Universal Robots URScript: 127765-201_OpticalBench_V1.script

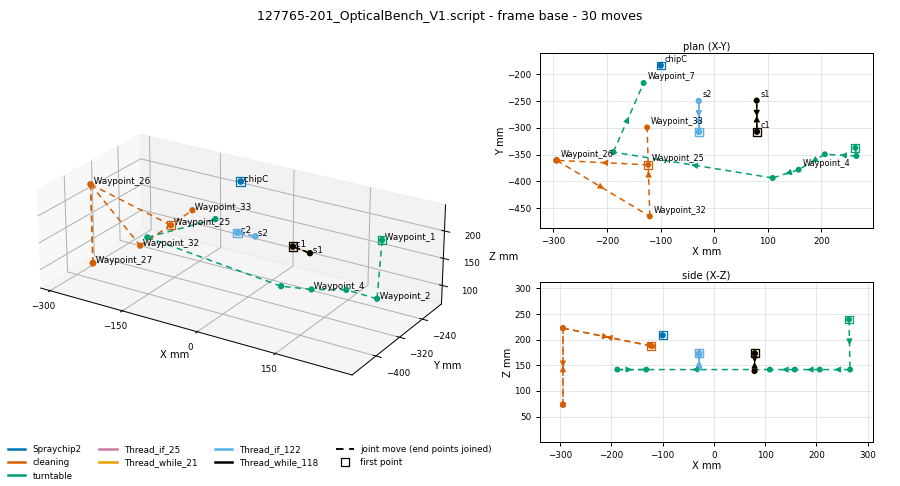
[picture p0: tool path of 127765-201_OpticalBench_V1.script in frame base, 30 of 121 moves have a stored position in this frame; points joined in program order, loops and branches not executed]
def P127765201_OpticalBench_V1():
  global _hidden_verificationVariable=0
  step_count_28707e12_0c2a_4f39_b822_8a6eb026eba7 = 0.0
  thread Step_Counter_Thread_bc455d1c_3720_4032_8e16_f4a00f067eee():
    while (True):
      step_count_28707e12_0c2a_4f39_b822_8a6eb026eba7 = step_count_28707e12_0c2a_4f39_b822_8a6eb026eba7 + 1.0
      sync()
    end
  end
  run Step_Counter_Thread_bc455d1c_3720_4032_8e16_f4a00f067eee()
  set_target_payload(0.530000, [0.009000, -0.039000, 0.092000], [0.000534, 0.000534, 0.000534, 0.000000, 0.000000, 0.000000])
  set_safety_mode_transition_hardness(1)
  set_tcp(p[0.0,0.0,0.11,0.0,0.0,0.0])
  set_tool_communication(False, 115200, 0, 1, 1.5, 3.5)
  set_tool_output_mode(0)
  set_tool_digital_output_mode(0, 1)
  set_tool_digital_output_mode(1, 1)
  set_tool_voltage(0)
  set_gravity([0.0, 0.0, 9.82])
  set_standard_analog_input_domain(0, 1)
  set_standard_analog_input_domain(1, 1)
  set_tool_analog_input_domain(0, 1)
  set_tool_analog_input_domain(1, 1)
  set_analog_outputdomain(0, 0)
  set_analog_outputdomain(1, 0)
  set_input_actions_to_default()
  global Al_plate=p[0.12405209206180495,-0.2666666051843552,0.020008101224669964,-9.276623980477388E-5,1.8107917580596192E-5,3.1233857134705927]
  global Frame2x2=p[0.18266245434305164,-0.34273121659514855,0.026002571110600767,-2.225423529876215E-4,3.0110667546023537E-4,3.1233976058306383]
  global Plane_1=p[0.0,0.0,0.0,0.0,0.0,0.0]
  global URlogoTutorial=p[-0.08178353973148575,-0.3363174165299142,0.04788621506469384,-3.9746155723688456E-5,-3.4682148779121894E-5,-1.5668291789091222]
  global carousel=p[0.13865255139760183,-0.25132593351268107,0.051531504137083003,-4.453572132438073E-5,-1.3071222590669835E-4,-3.1349676625391965]
  global carouselrod=p[0.2020731702281844,-0.34951442511341274,0.1947611446273096,3.139766958234101,-0.10689428010274801,-1.1796370330365635E-5]
  global paper=p[-0.09670794781244417,-0.3283412964648025,0.027665994240809913,-3.2057893450593004E-5,2.867088716161181E-5,-1.6085327915291054]
  global rod=p[0.13368013097420872,-0.41123185103490206,0.09926814901395645,2.2214229924093103,-2.2214158162465862,-2.9165882738638143E-5]
  # begin: URCap Installation Node
  #   Source: Remote TCP & Toolpath, 1.3.0.build16, Universal Robots A/S
  #   Type: Remote TCP & Toolpath
  mc_check_divergence = True
  mc_lookahead = 0.03
  mc_gain = 2000
  mc_dt = 0.004

  mc_conv_tol_s = 0.001
  mc_conv_loops = 100

  mc_ee_set_id = 2

  MC_GROUP_STANDBY = 0
  MC_GROUP_STOPPING = 2
  MC_GROUP_ERROR_STOP = 3

  MC_ERROR_PATHDIVERGED = 0
  MC_ERROR_COLLISION = 1
  MC_ERROR_JOINTLIMIT = 2
  MC_ERROR_SINGULARITY = 4
  MC_ERROR_PLANNINGFAILED = 16
  MC_ERROR_DAEMONSTOPPED = 1024
  MC_ERROR_SERVER_BUSY = 1025
  MC_ERROR_NOT_INITIALIZED = 2000

  MC_TOOLPATH_ERROR_NONE = 0
  MC_TOOLPATH_ERROR_FILELOAD = 1
  MC_TOOLPATH_ERROR_PARSE = 2
  MC_TOOLPATH_ERROR_EMPTYTOOLPATH = 3
  MC_TOOLPATH_ERROR_UNSUPPORTEDTYPE = 4

  MC_GROUP_STATUS_INPUT = 24
  MC_CURRENT_MOTION_ID_INPUT = 25
  MC_ERROR_CODE_INPUT = 26
  MC_DIGITAL_OUTPUTS_INPUT = 27
  MC_JOINT_VALUE_INPUT = 24
  MC_WATCHDOG_INPUT = 30
  MC_PATH_SPEED_INPUT = 31
  MC_SPEEDFACTOR_OUTPUT = 24

  mc_last_watchdog = 0
  mc_watchdog_counter = 0
  mc_watchdog_counter_limit = 100

  mc_last_motion_id = -1
  mc_group_status = MC_GROUP_STOPPING
  mc_server_started = False
  mc_rtcp_moving = False
  mc_debug_msg = False
  mc_gmm_initialized = False
  mc_last_digital_outputs = 0

  def mc_initialize(mode, tcp, doc=6):
  	mc_check_busy()

  	if (mode == 0 and doc == 6):
  		mc_ee_set_id = 0
  	end

  	if (mode == 1 and doc == 6):
  		mc_ee_set_id = 2
  	end

  	if (mode == 0 and doc == 5):
  		mc_ee_set_id = 1
  	end

  	if (mode == 1 and doc == 5):
  		mc_ee_set_id = 3
  	end

  	mc_initialize_internal(tcp)
  end

  def mc_initialize_internal(tcp):
  	if (mc_server_started == False):
  		global mc_server = rpc_factory("xmlrpc", "127.0.0.1:7828")
  		mc_server_started = True
  	end

  	mc_server.setDataStoreBoolean("IS_ON", "/robot/check_divergence", mc_check_divergence)
  	mc_server.reset()
  	mc_group_status = MC_GROUP_STANDBY
  	mc_set_speed_factor(1.0)
  	mc_server.setKinTransform(mc_ee_set_id, 0, tcp)
  	mc_gmm_initialized = False
  end

  def mc_check_busy():
  	enter_critical
  	if (mc_rtcp_moving == False):
  		mc_rtcp_moving = True
  	else:
  		mc_error_stop("", "", MC_ERROR_SERVER_BUSY)
  	end
  	exit_critical
  end

  def mc_add_linear(pose, a, v, r):
  	mc_check_ready()
  	ee_id = 0
  	buffer_mode = "BLENDING_NEXT"
  	transition_mode = "CORNER_DISTANCE"
  	id = mc_server.moveLinearAbsolute(pose, mc_ee_set_id, ee_id, v, a, buffer_mode, transition_mode, r)

  	if (id == -1):
  		mc_error_stop("Compute node returned ID ", id)
  	end

  	mc_last_motion_id = id

  	return id
  end

  def mc_add_circular(pose_via, pose_to, a, v, r, mode = 0):
  	mc_check_ready()
  	ee_id = 0
  	buffer_mode = "BLENDING_NEXT"
  	transition_mode = "CORNER_DISTANCE"
  	id = mc_server.moveCircularBorderAbsolute(pose_via, pose_to, mode, mc_ee_set_id, ee_id, v, a, buffer_mode, transition_mode, r)

  	if (id == -1):
  		mc_error_stop("Compute node returned ID ", id)
  	end

  	mc_last_motion_id = id

  	return id
  end

  def mc_add_path(path_id, a, v, r):
  	mc_check_ready()
  	ee_id = 0
  	buffer_mode = "BLENDING_NEXT"
  	transition_mode = "CORNER_DISTANCE"
  	id = mc_server.movePath(path_id, mc_ee_set_id, ee_id, v, a, buffer_mode, transition_mode, r)

  	if (id == -1):
  		result = mc_server.getErrorCode()
  		mc_toolpath_error_stop(result[0], result[1])
  	end

  	mc_last_motion_id = id

  	return id
  end

  def mc_load_path(nc_file, use_feedrate = False):
  	id = mc_server.loadPath(nc_file, use_feedrate)

  	if (id < 0):
  		result = mc_server.getErrorCode()
  		mc_toolpath_error_stop(result[0], result[1])
  	end

  	return id
  end

  def mc_get_target_rtcp_speed():
  	return read_input_float_register(MC_PATH_SPEED_INPUT)
  end

  def mc_check_ready():
  	if mc_group_status != MC_GROUP_STANDBY:
  		mc_error_stop("", "", MC_ERROR_NOT_INITIALIZED)
  	end
  end

  def mc_set_pcs(pcs):
  	ee_id = 0
  	mc_server.setCoordinateTransform(mc_ee_set_id, ee_id, pcs, "ABORTING")
  end

  def mc_set_digital_outputs():
  	current_do = read_input_integer_register(MC_DIGITAL_OUTPUTS_INPUT)
  	current_do_bin = integer_to_binary_list(current_do)
  	last_do_bin = integer_to_binary_list(mc_last_digital_outputs)
  	loopcounter = 0
  	while (loopcounter < 4):
  		value_bit = loopcounter * 6
  		port_bit_0 = value_bit + 1
  		port_bit_1 = value_bit + 2
  		port_bit_2 = value_bit + 3
  		port_bit_3 = value_bit + 4
  		port_bit_4 = value_bit + 5
  		last_port = binary_list_to_integer([last_do_bin[port_bit_0], last_do_bin[port_bit_1], last_do_bin[port_bit_2], last_do_bin[port_bit_3], last_do_bin[port_bit_4]])
  		current_port = binary_list_to_integer([current_do_bin[port_bit_0], current_do_bin[port_bit_1], current_do_bin[port_bit_2], current_do_bin[port_bit_3], current_do_bin[port_bit_4]])
  		if (current_port != 0 and (current_port != last_port or current_do_bin[value_bit] != last_do_bin[value_bit])):
  			if (current_port <= 8):
  				set_standard_digital_out(current_port - 1, current_do_bin[value_bit])
  			elif (current_port <= 16):
  				set_configurable_digital_out(current_port - 9, current_do_bin[value_bit])
  			else:
  				set_tool_digital_out(current_port - 17, current_do_bin[value_bit])
  			end
  		end
  		loopcounter = loopcounter + 1
  	end
  	mc_last_digital_outputs = current_do
  end

  def mc_run_motion(id=-1):
  	if (id == -1):
  		id = mc_last_motion_id
  	end

  	mc_debugMsg("Waiting for ID ", id)

  	if (mc_gmm_initialized == False):
  		mc_initialize_gmm()
  	end

  	mc_current_motion_id = read_input_integer_register(MC_CURRENT_MOTION_ID_INPUT)
  	mc_group_status = read_input_integer_register(MC_GROUP_STATUS_INPUT)
  	joint_targets = get_actual_joint_positions()
  	while (mc_current_motion_id <= id and mc_current_motion_id != -2 and mc_group_status != MC_GROUP_STOPPING and mc_group_status != MC_GROUP_ERROR_STOP):
  		mc_current_motion_id = read_input_integer_register(MC_CURRENT_MOTION_ID_INPUT)
  		mc_group_status = read_input_integer_register(MC_GROUP_STATUS_INPUT)

  		joint_targets = mc_get_joint_targets(joint_targets)
  		servoj(joint_targets, t = mc_dt, lookahead_time = mc_lookahead, gain = mc_gain)

  		mc_set_digital_outputs()

  		mc_check_watchdog()
  	end

  	if (mc_group_status == MC_GROUP_STOPPING or mc_group_status == MC_GROUP_ERROR_STOP):
  		stopj(45)

  		mc_debugMsg("Stopping due to error after ID ", id)

  		mc_server.setDataStoreBoolean("IS_RTCP_RUNNING", "/group_motion_manager", False)

  		error_code = read_input_integer_register(MC_ERROR_CODE_INPUT)
  		mc_error_stop("Compute node returned group status ", mc_group_status, error_code)

  		mc_rtcp_moving = False
  		mc_group_status = MC_GROUP_STOPPING
  	end

  	if (id == mc_last_motion_id):
  		mc_debugMsg("Stopping after ID ", id)
  		mc_check_convergence(joint_targets)

  		mc_server.setDataStoreBoolean("IS_RTCP_RUNNING", "/group_motion_manager", False)

  		mc_rtcp_moving = False
  		mc_group_status = MC_GROUP_STOPPING
  	end

  	mc_debugMsg("Completed ID ", id)
  end

  def mc_set_speed_factor(s):
  	write_output_float_register(MC_SPEEDFACTOR_OUTPUT, s)
  end

  def mc_initialize_gmm():
  	mc_current_motion_id = read_input_integer_register(MC_CURRENT_MOTION_ID_INPUT)
  	while (mc_current_motion_id != -1):
  		mc_current_motion_id = read_input_integer_register(MC_CURRENT_MOTION_ID_INPUT)
  		sleep(mc_dt)
  		mc_check_watchdog()
  	end

  	mc_server.setDataStoreBoolean("IS_RTCP_RUNNING", "/group_motion_manager", True)

  	while (mc_current_motion_id == -1):
  		mc_current_motion_id = read_input_integer_register(MC_CURRENT_MOTION_ID_INPUT)
  		sleep(mc_dt)
  		mc_check_watchdog()
  	end

  	mc_gmm_initialized = True
  end

  def mc_check_convergence(joint_targets):
  	loopcounter = 0
  	converged = False
  	while (converged == False and loopcounter < mc_conv_loops):

  		joint_targets = mc_get_joint_targets(joint_targets)
  		ur_targets = get_target_joint_positions()
  		joint_speeds = get_actual_joint_speeds()

  		position_converged = joint_targets[0] == ur_targets[0] and joint_targets[1] == ur_targets[1] and joint_targets[2] == ur_targets[2] and joint_targets[3] == ur_targets[3] and joint_targets[4] == ur_targets[4] and joint_targets[5] == ur_targets[5]
  		speed_converged = joint_speeds[0] <= mc_conv_tol_s and joint_speeds[1] <= mc_conv_tol_s and joint_speeds[2] <= mc_conv_tol_s and joint_speeds[3] <= mc_conv_tol_s and joint_speeds[4] <= mc_conv_tol_s and joint_speeds[5] <= mc_conv_tol_s
  		converged = position_converged and speed_converged

  		servoj(joint_targets, t = mc_dt, lookahead_time = mc_lookahead, gain = mc_gain)

  		loopcounter = loopcounter + 1
  	end

  	mc_debugMsg("Convergence loop count: ", loopcounter)
  end

  def mc_check_watchdog():
  	current_watchdog = read_input_float_register(MC_WATCHDOG_INPUT)

  	if (current_watchdog > mc_last_watchdog):
  		mc_last_watchdog = current_watchdog
  		mc_watchdog_counter = 0
  	else:
  		mc_watchdog_counter = mc_watchdog_counter + 1
  		if (mc_watchdog_counter > mc_watchdog_counter_limit):
  			mc_error_stop("", "", MC_ERROR_DAEMONSTOPPED)
  		end
  	end
  end

  def mc_get_joint_targets(joint_targets):
  	joint_targets[0] = read_input_float_register(MC_JOINT_VALUE_INPUT)
  	joint_targets[1] = read_input_float_register(MC_JOINT_VALUE_INPUT + 1)
  	joint_targets[2] = read_input_float_register(MC_JOINT_VALUE_INPUT + 2)
  	joint_targets[3] = read_input_float_register(MC_JOINT_VALUE_INPUT + 3)
  	joint_targets[4] = read_input_float_register(MC_JOINT_VALUE_INPUT + 4)
  	joint_targets[5] = read_input_float_register(MC_JOINT_VALUE_INPUT + 5)
  	return joint_targets
  end

  def mc_error_stop(msg, param="", error_code=MC_ERROR_PLANNINGFAILED):
  	if (msg != ""):
  		textmsg(msg, param)
  	end

  	textmsg("Error code: ", error_code)
  	error_msg = mc_getErrorMessage(error_code)
  	textmsg(error_msg)

  	popup(error_msg, title="Remote TCP", error=True, blocking=False)
  	halt
  end

  def mc_toolpath_error_stop(error_code, param):
  	msg = mc_getToolpathMessage(error_code)
  	textmsg(msg + " - Line: ", param)

  	popup(msg, title="Toolpath Validation", error=True, blocking=True)
  	halt
  end

  def mc_debugMsg(msg, param=""):
  	if (mc_debug_msg == True):
  		textmsg(msg, param)
  	end
  end
  def mc_getErrorMessage(error_code):
  	if error_code == MC_ERROR_PATHDIVERGED:
  		return "<html>Robot cannot maintain tool speed. You may avoid this issue by:<ul><li>reducing the tool speed;</li><li>avoiding sharp corners;</li><li>staying away from singularities.</li></ul></html>"
  	elif error_code == MC_ERROR_COLLISION:
  		return "Robot is in collision."
  	elif error_code == MC_ERROR_JOINTLIMIT:
  		return "Robot is at a joint limit."
  	elif error_code == MC_ERROR_SINGULARITY:
  		return "Robot is at a singularity."
  	elif error_code == MC_ERROR_DAEMONSTOPPED:
  		return "The controller stopped."
  	elif error_code == MC_ERROR_SERVER_BUSY:
  		return "Another Remote TCP Move node is running."
  	elif error_code == MC_ERROR_NOT_INITIALIZED:
  		return "Group motion manager is not initialized."
  	else:
  		return "Motion planning failed."
  	end
  end

  def mc_getToolpathMessage(message_code):
  	if message_code == MC_TOOLPATH_ERROR_NONE:
  		return "Toolpath file is valid."
  	elif message_code == MC_TOOLPATH_ERROR_FILELOAD:
  		return "File cannot be loaded."
  	elif message_code == MC_TOOLPATH_ERROR_PARSE:
  		return "Parsing error"
  	elif message_code == MC_TOOLPATH_ERROR_EMPTYTOOLPATH:
  		return "Empty toolpath"
  	elif message_code == MC_TOOLPATH_ERROR_UNSUPPORTEDTYPE:
  		return "Unsupported type"
  	else:
  		return "Unknown toolpath validation error"
  	end
  end
  # end: URCap Installation Node
  # begin: URCap Installation Node
  #   Source: Robotiq_Copilot, 2.7.0.56387, Robotiq Inc.
  #   Type: Machine Tending
  def rq_is_stack_light_machine_state_running():
    return False
  end
  def rq_is_stack_light_machine_state_idle():
    return False
  end
  # end: URCap Installation Node
  # begin: URCap Installation Node
  #   Source: Robotiq_Copilot, 2.7.0.56387, Robotiq Inc.
  #   Type: Copilot
  ###############################################################
  # Script file used to communicate with Robotiq's ft sensor
  # Version: 0.0.1
  ###############################################################

  node_rpc_server = rpc_factory("xmlrpc","http://127.0.0.1:4251/node")
  linalg = rpc_factory("xmlrpc","http://127.0.0.1:4251/linalg")
  storevar = rpc_factory("xmlrpc","http://127.0.0.1:4251/storevariable")
  kinematics_rpc_server = rpc_factory("xmlrpc","http://127.0.0.1:4251/")

  global Fx = 0.0
  global Fy = 0.0
  global Fz = 0.0
  global Mx = 0.0
  global My = 0.0
  global Mz = 0.0
  global T_base_sensor = p[0,0,0,0,0,0]
  global tcp_wrench = [0,0,0,0,0,0]
  global base_wrench = [0,0,0,0,0,0]
  global sensor_wrench = [0,0,0,0,0,0]
  global rq_depal_end_pose_offset = p[0,0,0,0,0,0]
  global rq_ft_sensor_connected = False

  rq_target_joint_positions = get_actual_joint_positions()
  rq_elapsed_time = 0
  rq_force_protect_urcap = 0.0
  rq_torque_protect_urcap = 0.0
  rq_collision_detection_enabled = False
  rq_collision_detection_active_time = 0.0
  rq_halt_on_collision_detection = True
  is_rq_prevent_steady_enabled = True
  rq_active_node = 0
  rq_node_executor_thread_running = False
  rq_lookahead_time = 0.05
  rq_continue_node_execution = True
  rq_controller_time_step = 0.008

  rq_linear_axis_move_abs_target_position = 0.0
  rq_linear_axis_move_abs_target_speed = 0.0 # Documented in monorepo/doc/pal/PalAdvancedProgrammingFunctions.md
  rq_linear_axis_move_abs_target_acc = 0.0 # Documented in monorepo/doc/pal/PalAdvancedProgrammingFunctions.md
  rq_linear_axis_move_abs_target_decel = 0.0 # Documented in monorepo/doc/pal/PalAdvancedProgrammingFunctions.md
  rq_linear_axis_move_absolute_thread = 0
  rq_linear_axis_move_absolute_thread_running = False

  def pose_to_list(p):
    return [p[0], p[1], p[2], p[3], p[4], p[5]]
  end

  def list_to_pose(l):
    return p[l[0], l[1], l[2], l[3], l[4], l[5]]
  end

  def rq_init_path(pathId):
     initPathAnswer = node_rpc_server.initpath(pathId)
     verify_path_answer(initPathAnswer)
     return initPathAnswer[0]
  end

  def concat(str1, str2, str3):
    return str_cat(str1, str_cat(str2, str3))
  end
  def key_val(key, val):
    return concat(concat("`", key, "`"), ":", val)
  end

  thread rq_prevent_steady():
    local q_start = get_target_joint_positions()
    local q = q_start
    local p = 0

    while True:
      p = p + rq_controller_time_step*4*3.14159
      local offset = 0.000001*sin(p)
      q[5] = q_start[5] + offset
      servoj(q)
    end
  end

  def linear_axis_move_abs(target_position,
                           target_speed,
                           target_acceleration,
                           target_deceleration,
                           is_blocking,
                           prevent_steady = True):
    rq_linear_axis_move_abs_target_position = target_position
    rq_linear_axis_move_abs_target_speed = target_speed
    rq_linear_axis_move_abs_target_acc = target_acceleration
    rq_linear_axis_move_abs_target_decel = target_deceleration
    is_rq_prevent_steady_enabled = prevent_steady

    if( rq_linear_axis_move_absolute_thread_running ):
      kill rq_linear_axis_move_absolute_thread
    end
    rq_linear_axis_move_absolute_thread = run linear_axis_move_abs_thread()
    if(is_blocking):
      join rq_linear_axis_move_absolute_thread
    end
  end #linear_axis_move_abs

  thread linear_axis_move_abs_thread():

    if is_rq_prevent_steady_enabled:
      rq_prevent_steady_thread = run rq_prevent_steady()
    end

    rq_linear_axis_move_absolute_thread_running = True
    timeout_in_milliseconds = 500
    target_position_reached = False
    number_of_done_status_received_while_not_at_target = 0

    while( not target_position_reached ):
      move_absolute_response = node_rpc_server.linearaxismove(rq_linear_axis_move_abs_target_position,
                                                              rq_linear_axis_move_abs_target_speed,
                                                              rq_linear_axis_move_abs_target_acc,
                                                              rq_linear_axis_move_abs_target_decel,
                                                              timeout_in_milliseconds)

      if move_absolute_response == 0: # Done
        position_tolerance = 1e-3
        local position = node_rpc_server.linearaxisgetactualposition() # local because it is a variable under 15 chars that a user could have defined
        target_position_reached = ( norm( position - rq_linear_axis_move_abs_target_position ) < position_tolerance )
        if not target_position_reached:
          number_of_done_status_received_while_not_at_target = number_of_done_status_received_while_not_at_target + 1
          if ( number_of_done_status_received_while_not_at_target > 10 ): #When the move starts, it may take some time before the status changes from done to busy so we accept a certain number of done status without being at the target position
            textmsg("error: target position should be reached when move absolute status is Done")
          end
        end
      elif move_absolute_response == 1: # Normal (safeguard stopped, busy moving, or paused)
        # do nothing
      elif move_absolute_response == 2: # Error
        textmsg("Linear axis absolute move error")
        popup("Program paused because axis is not ready or the requested position is outside the allowed range.",
              title="Linear axis move error", warning=False, error=True, blocking=True)
        socket_send_line("pause", "RQDashboardClient") # If the axis is not ready, this allows the user to go fix it and then resume the program.
        sleep(1.0) # The socket_send_line command is non-blocking, so we need to wait for the progam to pause.
                   # Without the sleep, execution will continue and multiple popups and program pauses will be executed.
      end

      sleep(rq_controller_time_step)
    end #while
    rq_linear_axis_move_absolute_thread_running = False

    if is_rq_prevent_steady_enabled:
      kill rq_prevent_steady_thread
    end

  end # linear_axis_move_abs_thread

  def setup_force_node_on_server(generic_rq_insertion_force_node_id = 1,
                                 feature=1,
                                 targetforce = [0,0,0,0,0,0],
                                 force_control_enabled_axes = [False, False, False, False, False, False],
                                 max_negative_deviation_vector = [-0.1, -0.1, -0.1, -0.1, -0.1, -0.1],
                                 max_positive_deviation_vector = [0.1, 0.1, 0.1, 0.1, 0.1, 0.1],
                                 adaptiveStiffness = True):
    node_rpc_server.setforcecontrolfeature(generic_rq_insertion_force_node_id, feature)
    node_rpc_server.setforcecontroltargetforce(generic_rq_insertion_force_node_id, targetforce)
    node_rpc_server.setforcecontrolenabledaxes(generic_rq_insertion_force_node_id, force_control_enabled_axes)
    node_rpc_server.setforcecontrolmaximaldeviation(generic_rq_insertion_force_node_id, max_negative_deviation_vector, max_positive_deviation_vector)
    node_rpc_server.setforcecontroladaptivestiffnessenabledaxes(generic_rq_insertion_force_node_id, True)
  end

  def verify_path_answer(path_answer):
   initPathStatusCode = path_answer[1]
   handle_path_node_error_code(initPathStatusCode)
  end

  def handle_path_node_error_code(initPathStatusCode):
    if initPathStatusCode == -1:
      popup("Could not compute path with the selected options.", "Robotiq's FT Sensor", blocking=True, error=True)
    elif initPathStatusCode == 1:
      popup("Joint solution impossible. Change your starting position.", "Robotiq's FT Sensor", blocking=True, error=True)
    elif initPathStatusCode == 2:
      popup("Discontinuous path detected. Change your starting position.", "Robotiq's FT Sensor", blocking=True, error=True)
    elif initPathStatusCode == 3:
      popup("Path time limit has been reached. Increase the speed of your path or break it down in multiple shorter paths.", "Robotiq's FT Sensor", blocking=True, error=True)
    elif initPathStatusCode == 4:
      popup("Could not compute path with the selected options. Computing path timeout.", "Robotiq's FT Sensor", blocking=True, error=True)
    elif initPathStatusCode == 5:
      popup("Path computation was aborted.", "Robotiq's FT Sensor", blocking=True, error=True)
    elif initPathStatusCode == 6:
      popup("A previous path computation is still in progress. Please try again in a few seconds.", "Robotiq's FT Sensor", blocking=True, error=True)
    elif initPathStatusCode == 7:
      textmsg("Path initialization error: Invalid path id.") # No popup needed in this case.
    elif initPathStatusCode == 8:
      popup("Palletizer error: box number out of range.", blocking=True, error=True)
    elif initPathStatusCode == 9:
      popup("Palletizer error: collision detected.", blocking=True, error=True)
    elif initPathStatusCode == 10:
      popup("Palletizer error: boxes overlap in layer.", blocking=True, error=True)
    elif initPathStatusCode == 11:
      popup("Palletizer error: empty layer.", blocking=True, error=True)
    elif initPathStatusCode == 12:
      popup("Palletizer error: The PLC was not connected during node creation.", blocking=True, error=True)
    elif initPathStatusCode != 0:
      textmsg("Unexpected initPathStatusCode value : ", initPathStatusCode)
    end

    if initPathStatusCode != 0:
      halt
    end
  end

  def rq_wait_ft_sensor_steady(timeout = 2000):

    max_mean_squared_error = [0.1, 0.1, 0.1, 0.0001, 0.0001, 0.0001]
    local mean = sensor_wrench

    mean_squared_error = sensor_wrench
    local i = 0
    while i<6:
      mean_squared_error[i] = mean_squared_error[i] * mean_squared_error[i]
      i=i+1
    end

    is_sensor_steady = False
    local alpha = 0.9
    local timer = 0

    while (not is_sensor_steady) and (timer < timeout):
      sleep(rq_controller_time_step)
      timer = timer + 8

      i = 0
      while i < 6:
        mean[i] = alpha * mean[i] + (1.0 - alpha) * sensor_wrench[i]
        error = sensor_wrench[i] - mean[i]
        mean_squared_error[i] = alpha * mean_squared_error[i] + ((1.0 - alpha) * error * error)
        i = i+1
      end

      is_sensor_steady = True
      i = 0
      while (i < 6) and is_sensor_steady:
        is_sensor_steady = mean_squared_error[i] < max_mean_squared_error[i]
        i = i+1
      end
    end

    return is_sensor_steady
  end

  thread rq_elapsed_timer_ms():
    rq_elapsed_time = 0
    dt = 1000/500
    while True:
      rq_elapsed_time =  rq_elapsed_time + dt
      sync()
    end
  end

  def get_sensor_fx():
    return Fx
  end

  def get_sensor_fy():
    return Fy
  end

  def get_sensor_fz():
    return Fz
  end

  def get_sensor_mx():
    return Mx
  end

  def get_sensor_my():
    return My
  end

  def get_sensor_mz():
    return Mz
  end

  def get_applied_tcp_force(index):
    return -1.0 * tcp_wrench[index]
  end

  def get_applied_base_force(index):
    return -1.0 * base_wrench[index]
  end

  def express_vector_in_new_frame(T_from_to, V_from):
    Q_from_to = p[0, 0, 0, T_from_to[3], T_from_to[4], T_from_to[5]]
    V_to = pose_trans(pose_inv(Q_from_to), p[V_from[0], V_from[1], V_from[2], 0, 0, 0])
    return [V_to[0], V_to[1], V_to[2]]
  end

  def express_force_in_frame(T_from_to, wrench_from):
    F = express_vector_in_new_frame(T_from_to, [wrench_from[0], wrench_from[1], wrench_from[2]])
    T = express_vector_in_new_frame(T_from_to, [wrench_from[3], wrench_from[4], wrench_from[5]])
    return [F[0], F[1], F[2], T[0], T[1], T[2]]
  end

  def express_pose_A_relative_to_pose_B(pose_A, pose_B):
    return pose_trans(pose_inv(pose_B), pose_A)
  end

  thread read_force():

    if (not socket_open("127.0.0.1", 29999, "RQDashboardClient")):
      popup("Can't connect to the Dashboard server", "Robotiq's FT Sensor", error=True)
      halt
    end

    rq_collision_detection_active_count = 0
    rq_collision_detection_active = False

    while True:
        T_base_tcp = get_actual_tcp_pose()
        T_base_flange = get_actual_tool_flange_pose()
        T_flange_sensor = p[0, 0, 0, 0, 0, 0]
        T_base_sensor = pose_trans(T_base_flange, T_flange_sensor)

        T_flange_tcp = pose_trans( pose_inv(T_base_flange), T_base_tcp)
        T_sensor_tcp = pose_trans( pose_inv(T_flange_sensor), T_flange_tcp)

        sensor_wrench = express_force_in_frame(T_base_sensor, get_tcp_force())
        tcp_wrench = wrench_trans(pose_inv(T_sensor_tcp), sensor_wrench)
        base_wrench = express_force_in_frame(pose_inv(T_base_tcp), tcp_wrench)

        Fx = sensor_wrench[0]
        Fy = sensor_wrench[1]
        Fz = sensor_wrench[2]
        Mx = sensor_wrench[3]
        My = sensor_wrench[4]
        Mz = sensor_wrench[5]

        write_output_float_register(TCP_FX_ACTUAL_OUTPUT_DOUBLE, tcp_wrench[0])
        write_output_float_register(TCP_FY_ACTUAL_OUTPUT_DOUBLE, tcp_wrench[1])
        write_output_float_register(TCP_FZ_ACTUAL_OUTPUT_DOUBLE, tcp_wrench[2])
        write_output_float_register(TCP_MX_ACTUAL_OUTPUT_DOUBLE, tcp_wrench[3])
        write_output_float_register(TCP_MY_ACTUAL_OUTPUT_DOUBLE, tcp_wrench[4])
        write_output_float_register(TCP_MZ_ACTUAL_OUTPUT_DOUBLE, tcp_wrench[5])

        if rq_collision_detection_enabled:
            if rq_collision_detection_active_time < (0.5*rq_controller_time_step):
                if norm([Fx, Fy, Fz]) > rq_force_protect_urcap:
                    rq_on_collision_detection("Force limit value exceeded.")
                elif norm([Mx, My, Mz]) > rq_torque_protect_urcap:
                    rq_on_collision_detection("Torque limit value exceeded.")
                end
            else:
                rq_collision_detection_active_time = rq_collision_detection_active_time + rq_controller_time_step
                if rq_collision_detection_active_time >= 1.0:
                    rq_collision_detection_active_time = 0.0
                end
            end
        end

        sync()
        sync()
        sync()
        sync()

    end
  end

  def rq_get_ft_sensor_state():
    socket_open("127.0.0.1",63350,"rq_ft_sensor_state")
    socket_send_string("CURRENT STATE", "rq_ft_sensor_state")
    rq_sensor_state = socket_read_string("rq_ft_sensor_state")
    socket_close("rq_ft_sensor_state")

    if rq_sensor_state == "":
      rq_sensor_state = "RQ_STATE_INIT"
    end

    return rq_sensor_state
  end

  def rq_ft_sensor_disconnected_warn_user():
    socket_open("127.0.0.1",29999,"SensorWarning")
    socket_send_string("popup FT Sensor must be connected to run this program.","SensorWarning")
    socket_send_byte(10,"SensorWarning")
    socket_close("SensorWarning")
  end

  def rq_ft_sensor_disconnected_stop_program():
    socket_open("127.0.0.1", 30002, "rq_ft_sensor_stop_socket")

    socket_send_string("def rq_ft_sensor_stop_program():", "rq_ft_sensor_stop_socket")
    socket_send_byte(10, "rq_ft_sensor_stop_socket")
    socket_send_string("  stopj(5.0)", "rq_ft_sensor_stop_socket")
    socket_send_byte(10, "rq_ft_sensor_stop_socket")
    socket_send_string("end", "rq_ft_sensor_stop_socket")
    socket_send_byte(10, "rq_ft_sensor_stop_socket")

    socket_close("rq_ft_sensor_stop_socket")
  end

  def rq_ft_sensor_disconnected_check():
    if rq_get_ft_sensor_state() == "RQ_STATE_INIT":
      rq_ft_sensor_disconnected_stop_program()
      rq_ft_sensor_disconnected_warn_user()

      return True
    else:
      return False
    end
  end

  #RTDE input registers
  TARGET_JOINT_0_INPUT_REGISTER_DOUBLE = 40
  TARGET_JOINT_1_INPUT_REGISTER_DOUBLE = 41
  TARGET_JOINT_2_INPUT_REGISTER_DOUBLE = 42
  TARGET_JOINT_3_INPUT_REGISTER_DOUBLE = 43
  TARGET_JOINT_4_INPUT_REGISTER_DOUBLE = 44
  TARGET_JOINT_5_INPUT_REGISTER_DOUBLE = 45
  FINISH_NODE_INPUT_REGISTER_INT32 = 40
  RUNTIME_ERROR_INPUT_REGISTER_INT32 = 41
  ACTIVATION_NODE_COUNT_INPUT_REGISTER_INT32 = 42

  #RTDE output registers
  ACTIVE_NODE_OUTPUT_REGISTER_INT32 = 40
  NODE_EXECUTION_OUTPUT_COUNT_INT32 = 41
  ACTIVATION_NODE_COUNT_OUTPUT_REGISTER_INT32 = 42
  TCP_FX_ACTUAL_OUTPUT_DOUBLE = 34
  TCP_FY_ACTUAL_OUTPUT_DOUBLE = 35
  TCP_FZ_ACTUAL_OUTPUT_DOUBLE = 36
  TCP_MX_ACTUAL_OUTPUT_DOUBLE = 37
  TCP_MY_ACTUAL_OUTPUT_DOUBLE = 38
  TCP_MZ_ACTUAL_OUTPUT_DOUBLE = 39
  GENERAL_OUTPUT_DOUBLE_40 = 40
  GENERAL_OUTPUT_DOUBLE_41 = 41
  GENERAL_OUTPUT_DOUBLE_42 = 42
  GENERAL_OUTPUT_DOUBLE_43 = 43
  GENERAL_OUTPUT_DOUBLE_44 = 44
  GENERAL_OUTPUT_DOUBLE_45 = 45

  write_output_integer_register(ACTIVE_NODE_OUTPUT_REGISTER_INT32, 0)
  write_output_integer_register(NODE_EXECUTION_OUTPUT_COUNT_INT32, 0)
  write_output_integer_register(ACTIVATION_NODE_COUNT_OUTPUT_REGISTER_INT32, 0)
  write_output_float_register(TCP_FX_ACTUAL_OUTPUT_DOUBLE, 0)
  write_output_float_register(TCP_FY_ACTUAL_OUTPUT_DOUBLE, 0)
  write_output_float_register(TCP_FZ_ACTUAL_OUTPUT_DOUBLE, 0)
  write_output_float_register(TCP_MX_ACTUAL_OUTPUT_DOUBLE, 0)
  write_output_float_register(TCP_MY_ACTUAL_OUTPUT_DOUBLE, 0)
  write_output_float_register(TCP_MZ_ACTUAL_OUTPUT_DOUBLE, 0)

  global activation_node_count = 0
  global node_execution_count = 0

  def element_wise_subtract(l1, l2):
    local r = l1
    local i = 0
    while i<length(r):
      r[i]=l1[i]-l2[i]
      i=i+1
    end
    return r
  end

  def element_wise_add(l1, l2):
    local result = l1
    local i = 0
    while i < length(result):
      result[i] = l1[i] + l2[i]
      i = i + 1
    end
    return result
  end

  def list_by_scalar_multiply(l1, scalar):
      local r = l1
      local i = 0
      while i<length(r):
        r[i]=l1[i]*scalar
        i=i+1
      end
      return r
   end

  def norm_inf(v):
    local norm = 0
    local i = 0
    while i<length(v):
        n = norm(v[i])
        if(n > norm):
          norm = n
        end
      i=i+1
    end
    return norm
  end

  def active_and_reset_node(nodeId):
    server_activation_node_count = read_input_integer_register(ACTIVATION_NODE_COUNT_INPUT_REGISTER_INT32)

    activation_node_count = activation_node_count + 1
    node_execution_count = 0
    write_output_integer_register(NODE_EXECUTION_OUTPUT_COUNT_INT32, node_execution_count)
    rq_active_node = nodeId
    write_output_integer_register(ACTIVE_NODE_OUTPUT_REGISTER_INT32, nodeId)
    write_output_integer_register(ACTIVATION_NODE_COUNT_OUTPUT_REGISTER_INT32, activation_node_count)

    while server_activation_node_count == read_input_integer_register(ACTIVATION_NODE_COUNT_INPUT_REGISTER_INT32):
      sleep(rq_controller_time_step)
    end
  end

  def execute_node(nodeId, startThread = False):
    node_execution_thread = 0
    active_and_reset_node(nodeId)
    if startThread:
      rq_target_joint_positions = get_actual_joint_positions()
      movej(rq_target_joint_positions) # This movej is used to prevent the "another thread is already controlling the robot" error.
      rq_continue_node_execution = True
      node_execution_thread = run execute_node_thread()
    end
    while not active_node_completed():
      sync()
    end
    return node_execution_thread
  end

  def setup_node_execution_related_variables():
    activation_node_count = 0
    node_execution_count = 0
    write_output_integer_register(ACTIVE_NODE_OUTPUT_REGISTER_INT32, 0)
    write_output_integer_register(ACTIVATION_NODE_COUNT_OUTPUT_REGISTER_INT32, activation_node_count)
    write_output_integer_register(NODE_EXECUTION_OUTPUT_COUNT_INT32, node_execution_count)
    sleep(rq_controller_time_step)
  end

  def start_node_executor():
    setup_node_execution_related_variables()

    succeeded = node_rpc_server.startnodeexecutor()
    if not succeeded:
      node_rpc_server.stopnodeexecutor()
      sleep(0.5) # Needed for URControl to free the input registers.
      succeeded = node_rpc_server.startnodeexecutor()
      if not succeeded:
        popup("RTDE interface cannot initialize. Make sure that Ethernet/IP adapter and Profinet are disabled, and that no other URCaps use the RTDE interface.", "Robotiq Copilot", error=True)
        halt
      end
    end

    hand_shake_xmlrpcserver()
  end

  def reset_node_executor():
    setup_node_execution_related_variables()

    succeeded = node_rpc_server.resetnodeexecutor()
    if not succeeded:
      popup("RTDE interface cannot initialize. Make sure that Ethernet/IP adapter and Profinet are disabled, and that no other URCaps use the RTDE interface.", "Robotiq Copilot", error=True)
      halt
    end

    hand_shake_xmlrpcserver()
  end

  def hand_shake_xmlrpcserver():
    timer_thread = run rq_elapsed_timer_ms()
    sleep(rq_controller_time_step)
    node_execution_initialized = False
    while (not node_execution_initialized) and (rq_elapsed_time < 100):
      node_execution_initialized = (read_input_integer_register(FINISH_NODE_INPUT_REGISTER_INT32) == -1)
      sleep(rq_controller_time_step)
    end
    kill timer_thread

    if (not node_execution_initialized):
      popup("Node Execution initialization failed.", "Robotiq Copilot", error=True)
      halt
    end
  end

  thread execute_node_thread():
    rq_target_joint_positions = get_actual_joint_positions()
    servoj(rq_target_joint_positions)
    while rq_continue_node_execution:
      new_rq_target_joint_positions = update_target_position()
      joint_target_distances = element_wise_subtract(new_rq_target_joint_positions, rq_target_joint_positions)
      max_joint_target_displacement = norm_inf(joint_target_distances)
      if max_joint_target_displacement > 0.2:
          textmsg("previous target position: ", rq_target_joint_positions)
          textmsg("next target position: ", new_rq_target_joint_positions)
          textmsg("max joint target displacement: ", max_joint_target_displacement)
          popup("Node executor error: see Log tab for details", "Robotiq Copilot", False, True, True)
          halt
      end

      local i = 1
      while i < 5: # (servoj frequency)/(rtde frequency) = 500/125 = 4
        rq_target_joint_positions_interpolated = element_wise_add( rq_target_joint_positions,
                                                                   list_by_scalar_multiply(joint_target_distances, 0.25*i) )
        servoj(rq_target_joint_positions_interpolated, t=get_steptime(), lookahead_time=rq_lookahead_time, gain=500)
        i = i + 1
      end

      rq_target_joint_positions = new_rq_target_joint_positions
    end
    stopj(5)
  end

  # The thread below is used to prevent "another thread is already controlling the robot error".
  # In some occasions, even a sleep(0.05) will not work so this is necessary (until fixed by UR).
  # The thread is immediately killed to avoid unnecessary motion for the case of a parent node
  # that modifies the servoj target joint positions.
  def kill_thread( thread_id ):
    kill thread_id
    run_movej_thread = run movej_thread()
    sleep(rq_controller_time_step)
    kill run_movej_thread
  end

  thread movej_thread():
    movej(rq_target_joint_positions)
  end

  def active_node_completed():
    return (read_input_integer_register(ACTIVATION_NODE_COUNT_INPUT_REGISTER_INT32) == activation_node_count) and
           (read_input_integer_register(FINISH_NODE_INPUT_REGISTER_INT32) == rq_active_node)
  end

  def rq_handle_error_code(code):
    message = "Runtime error!"

    if code == 1:
      message = "Robotiq license error!"
    elif code == 2:
      message = "Program stopped due to runtime error. Please restart the program."
    end

    popup(message, "Robotiq Copilot", error=True)
    halt
  end

  def update_target_position():

    error_code = read_input_integer_register(RUNTIME_ERROR_INPUT_REGISTER_INT32)

    if error_code != 0:
      rq_handle_error_code(error_code)
    end

    new_rq_target_joint_positions = [0,0,0,0,0,0]
    new_rq_target_joint_positions[0] = read_input_float_register(TARGET_JOINT_0_INPUT_REGISTER_DOUBLE)
    new_rq_target_joint_positions[1] = read_input_float_register(TARGET_JOINT_1_INPUT_REGISTER_DOUBLE)
    new_rq_target_joint_positions[2] = read_input_float_register(TARGET_JOINT_2_INPUT_REGISTER_DOUBLE)
    new_rq_target_joint_positions[3] = read_input_float_register(TARGET_JOINT_3_INPUT_REGISTER_DOUBLE)
    new_rq_target_joint_positions[4] = read_input_float_register(TARGET_JOINT_4_INPUT_REGISTER_DOUBLE)
    new_rq_target_joint_positions[5] = read_input_float_register(TARGET_JOINT_5_INPUT_REGISTER_DOUBLE)

    node_execution_count = node_execution_count + 1
    write_output_integer_register(NODE_EXECUTION_OUTPUT_COUNT_INT32, node_execution_count)
    return new_rq_target_joint_positions
  end

  def set_servoj_node_cmd(q):
    write_output_float_register(GENERAL_OUTPUT_DOUBLE_40, q[0])
    write_output_float_register(GENERAL_OUTPUT_DOUBLE_41, q[1])
    write_output_float_register(GENERAL_OUTPUT_DOUBLE_42, q[2])
    write_output_float_register(GENERAL_OUTPUT_DOUBLE_43, q[3])
    write_output_float_register(GENERAL_OUTPUT_DOUBLE_44, q[4])
    write_output_float_register(GENERAL_OUTPUT_DOUBLE_45, q[5])
  end

  def rq_collision_detection_start(force_limit = 140, torque_limit = 14, halt_on_collision = True):
    rq_force_protect_urcap = force_limit
    rq_torque_protect_urcap = torque_limit
    rq_collision_detection_active_time = 0.0
    rq_collision_detection_enabled = True
    rq_halt_on_collision_detection = halt_on_collision
  end

  def rq_collision_detection_stop():
    rq_collision_detection_enabled = False
  end

  def rq_on_collision_detection(message):
    textmsg("Collision Detection. " + message)
    popupTitle = "Collision Detection"
    if rq_halt_on_collision_detection:
      popup(message + " Program halt.", popupTitle, False, True, False)
      halt
    else:
      popup(message + " Program suspend.", popupTitle, True, False, False)
      socket_send_line("pause", "RQDashboardClient")
      rq_collision_detection_active_time = rq_controller_time_step
    end
  end

  def round(number_to_round):
    if number_to_round - floor(number_to_round) < 0.5:
      return floor(number_to_round)
    else:
      return ceil(number_to_round)
    end
  end

  # Documented in monorepo/doc/pal/PalAdvancedProgrammingFunctions.md
  def rq_execute_box_trajectory(nodeId, current_box_count, has_box_payload, end_pose_offset = p[0,0,0,0,0,0]):
    rq_lookahead_time = 0.08
    local payload_mass = get_target_payload()
    local payload_cog  = get_target_payload_cog()
    local flange_payload = [payload_mass, payload_cog[0], payload_cog[1], payload_cog[2]]

    path_answer = node_rpc_server.initboxtrajectory(nodeId, current_box_count, has_box_payload, flange_payload, end_pose_offset)

    verify_path_answer(path_answer)
    reset_node_executor()
    node_execution_thread = execute_node(nodeId, True)
    rq_continue_node_execution = False
    join node_execution_thread
    rq_lookahead_time = 0.05
  end

  ################################
  # MAIN
  ################################

  run read_force()
  start_node_executor()

  preparationErrorXmlRpcClient = rpc_factory("xmlrpc","http://localhost:45697")
  contactOffsetXmlRpcClient = rpc_factory("xmlrpc","http://localhost:41787")
  palletizerXmlRpcClient = rpc_factory("xmlrpc","http://localhost:46233")
  machineTendingXmlRpcClient = rpc_factory("xmlrpc","http://localhost:36739")
    ###############################################################
    # Halt if a script preparation error occurred
    ###############################################################
    def checkForScriptPreparationException():
      if(preparationErrorXmlRpcClient.hasErrorOccurred()):
        popup(preparationErrorXmlRpcClient.getErrorMessage(), title=preparationErrorXmlRpcClient.getNodeInErrorTitle(), error=True, blocking=True)
        halt
      end
    end

    checkForScriptPreparationException()
  #***********************************************************************************************
  # verify tap detection
  #***********************************************************************************************

  def rq_tap_count(forces, high_threshold):

    low_threshold = 2
    tapCount = 0
    lookingForPeak = True
    indexDown = 0

    i = 1
    lastIndex = length(forces) - 1
    while i <= lastIndex:

      deltaForce = forces[i] - forces[0]

     if lookingForPeak:
        if deltaForce >  high_threshold:
          lookingForPeak = False
        end
      else:
        if deltaForce < low_threshold:
          tapCount = tapCount + 1
          lookingForPeak = True
          indexDown = i
        end
      end
      i = i + 1

    end

    if indexDown != lastIndex:
      tapCount = 0
    end

    return tapCount

  end
  def shift_right(list, default_value = 0):

     i = length(list)-1
     while (i > 0):
        list[i]=list[i-1]
        i=i-1
     end
     list[0] = default_value

     return list
  end

  #***********************************************************************************************
  # Wait for force reached
  #***********************************************************************************************
  # desired_wrench : desired wrench
  # is_active      : list of 0 and 1, 1 : axis is controlled
  # feature        : 0:base, 1:tcp
  # timeout        : timeout in miliseconds
  #***********************************************************************************************
  def rq_wait_for_force_reached(desired_wrench, is_active, feature, timeout):

    feature_base = 0
    feature_tool = 1
    time_constant = 0.025
    alpha = 1 - pow(2.718, -1.0 * rq_controller_time_step / time_constant)

    thresholds = [0.0, 0.0, 0.0, 0.0, 0.0, 0.0]
    minimal_thresholds = [1.0, 1.0, 1.0, 0.1, 0.1, 0.1]

    applied_wrench = [0.0, 0.0, 0.0, 0.0, 0.0, 0.0]
    filtered_wrench = [0.0, 0.0, 0.0, 0.0, 0.0, 0.0]

    if (feature == feature_base):
      applied_wrench = list_by_scalar_multiply(base_wrench, -1.0)
    else:
      applied_wrench = list_by_scalar_multiply(tcp_wrench, -1.0)
    end
    filtered_wrench = applied_wrench

    i = 0
    while (i < 6):
      if (is_active[i]):
        thresholds[i] = 0.05 * norm(desired_wrench[i])
        if thresholds[i] < minimal_thresholds[i]:
          thresholds[i] = minimal_thresholds[i]
        end
      else:
        thresholds[i] = 10000
      end
      i = i+1
    end

   force_reached = False

   timer = 0

   while ((not force_reached) and (timer < timeout)):

      if (feature == feature_base):
         applied_wrench = list_by_scalar_multiply(base_wrench, -1.0)
      else:
         applied_wrench = list_by_scalar_multiply(tcp_wrench, -1.0)
      end

      i = 0
      while (i < 6):
        filtered_wrench[i] = (alpha * applied_wrench[i]) + ((1.0 - alpha) * filtered_wrench[i])
        i = i+1
      end

      force_reached = True

      i = 0
      while ((i < 6) and force_reached):
        error = norm(desired_wrench[i] - filtered_wrench[i])
        if (error > thresholds[i]):
          force_reached = False
        end
        i = i + 1
      end

      timer = timer + rq_controller_time_step

      sleep(rq_controller_time_step)

    end

    return force_reached
  end
  #***********************************************************************************************
  # verify click detection
  #***********************************************************************************************
  click_detection_children_ended = False

  def rq_click_detection(force_drop_threshold = 10, torque_drop_threshold = 1, force_radio_button_selected = True):

    current_norm = 0
    drop_threshold = 0
    norms = [0.0, 0.0, 0.0, 0.0, 0.0]
    click_detected = False
    wrench_indices = [0,0,0]

    if(force_radio_button_selected):
      drop_threshold = force_drop_threshold
      wrench_indices = [0,1,2]
    else:
      drop_threshold =torque_drop_threshold
      wrench_indices = [3,4,5]
    end

    while ((not click_detection_children_ended) and (not click_detected)):

      current_norm = norm([sensor_wrench[wrench_indices[0]], sensor_wrench[wrench_indices[1]], sensor_wrench[wrench_indices[2]]])

      norms[4] = norms[3]
      norms[3] = norms[2]
      norms[2] = norms[1]
      norms[1] = norms[0]
      norms[0] = current_norm

      avg_norm = (norms[2] + norms[3] + norms[4]) / 3.0

      #Check if clicking is detected with force
      norm_drop = avg_norm - current_norm
      if(norm_drop > drop_threshold):
        textmsg("Click detected")
        click_detected=True
      else:
        sleep(rq_controller_time_step)
      end
    end

    return click_detected
  end
  ###############################################################
  # Script file used to define Robotiq functions for the Insertion node
  # Version: 0.0.2
  ###############################################################

  rq_ins_offset = p[0, 0, 0, 0, 0, 0]
  rq_ins_start_pose = p[0, 0, 0, 0, 0, 0]
  rq_actual_to_destination = p[0, 0, 0, 0, 0, 0]
  rq_ins_destination =p[0, 0, 0, 0, 0, 0]
  rq_ins_speed_setting = 0
  rq_rotation_not_completed = False
  rq_find_bottom_not_completed = False
  rq_spiral_not_completed = False

  def ins_actual_force_urcap(direction="X+"):
    axis = str_at(direction, 0)
    if (axis == "x") or (axis == "X"):
      return norm(get_applied_tcp_force(0))
    elif (axis == "y") or (axis == "Y"):
      return norm(get_applied_tcp_force(1))
    elif (axis == "z") or (axis == "Z"):
      return norm(get_applied_tcp_force(2))
    else:
      textmsg("ins_actual_force_urcap, invalid direction ", direction)
    end
  end

  def ins_actual_torque_urcap(direction = "Z+"):
    if (direction == "X+") or (direction == "X-") or (direction == "X"):
      return get_applied_tcp_force(3)
    elif (direction == "Y+") or (direction == "Y-") or (direction == "Y"):
      return get_applied_tcp_force(4)
    else:
      return get_applied_tcp_force(5)
    end

  end

  def square(a):
    return a*a
  end

  def update_servoj_node_target(target_joint_pos):
    set_servoj_node_cmd(target_joint_pos)
    sleep(rq_controller_time_step)
  end

  def create_all_insertion_nodes():
    global rq_insertion_force_node_id = node_rpc_server.createnewforcenode()
    global rq_insertion_movej_node_id = node_rpc_server.createnewmovejnode()
    global rq_insertion_servoj_node_id = node_rpc_server.createnewservojnode()
    node_rpc_server.setparentid(rq_insertion_movej_node_id, rq_insertion_force_node_id)
    node_rpc_server.setparentid(rq_insertion_servoj_node_id, rq_insertion_force_node_id)
  end

  def get_offset_projected_in_spiral_plane(direction, current_pose, pose_ref):
    axis = str_at(direction, 0)
    axis_index = 0
    if axis == "X":
      axis_index = 0
    elif axis == "Y":
      axis_index = 1
    elif axis == "Z":
      axis_index = 2
    else:
      textmsg("get_offset_projected_in_spiral_plane, invalid direction ", direction)
    end

    pose_offset = pose_trans( pose_inv(pose_ref), current_pose ) # current_pose and pose_ref should have the same orientations.
                                                                 # pose_offset is returned expressed in pose_ref frame

    pose_offset[axis_index] = 0 # valeur en direction mise a zero
    pose_offset[3] = 0 # valeur en Rx mise a zero
    pose_offset[4] = 0 # valeur en Ry mise a zero
    pose_offset[5] = 0 # valeur en Rz mise a zero

    return pose_offset
  end

  def update_spiral_offset(direction, spiral_initial_pose, spiral_initial_pose_offset, spiral_initial_pose_offset_name):
    pos_diff_tcp = get_offset_projected_in_spiral_plane(direction, get_actual_tcp_pose(), spiral_initial_pose)
    spiral_initial_pose_offset = interpolate_pose(spiral_initial_pose_offset, pos_diff_tcp, 0.35)
    storevar.setvariablepose(spiral_initial_pose_offset_name, spiral_initial_pose_offset)
  end

  def determine_max_spiral_radius_from_actual_position(direction, spiral_initial_pose, max_radius):
      dist_to_initial_pose = norm( get_offset_projected_in_spiral_plane(direction, get_actual_tcp_pose(), spiral_initial_pose))
      if (max_radius > dist_to_initial_pose):
        new_max_radius = max_radius - dist_to_initial_pose
      else:
        new_max_radius = 0
      end

      return new_max_radius
  end

  def insertion_compliant_move_urcap(axis = "Z",
                                     direction_sign = 1,
                                     compliant_insert_force_threshold = 20,
                                     speed = 0.04,
                                     feature = 1,
                                     max_position_deviation = 0.1):
    feature_base = 0
    feature_tool = 1

    if axis == "X":
      axis_index = 0
    elif axis == "Y":
      axis_index = 1
    elif axis == "Z":
      axis_index = 2
    else:
      textmsg("insertion_compliant_move_urcap, invalid direction ", axis)
    end

    current_pose = get_actual_tcp_pose()
    insertion_offset = p[0,0,0,0,0,0]
    rq_actual_to_destination = pose_trans(pose_inv(current_pose), rq_ins_destination)
    insertion_offset[axis_index] = rq_actual_to_destination[axis_index]
    insertion_pose = pose_trans(current_pose, insertion_offset)
    distance = point_dist(current_pose, insertion_pose)
    number_of_steps = floor( distance / (speed * rq_controller_time_step) ) + 1
    alpha_step  = 1.0 / number_of_steps

    # initialize forcenode
    node_execution_thread = initialise_force_node(position_controlled_direction = axis_index,
                                                  feature = feature_tool,
                                                  max_position_deviation = max_position_deviation)

    alpha = 0.0
    surface_found = False
    while (alpha <= 1.0) and (not surface_found):
      alpha = alpha + alpha_step
      interpolated_pose = interpolate_pose(current_pose, insertion_pose, alpha)
      q0 = get_inverse_kin(interpolated_pose) # define waypoint target
      update_servoj_node_target(q0)
      force = 0
      if feature == feature_base:
        force = get_applied_base_force(axis_index)
      elif feature == feature_tool:
        force = get_applied_tcp_force(axis_index)
      end
      if (direction_sign * force) >= compliant_insert_force_threshold:
        surface_found = True
      end
    end

    final_pos_reached = (alpha >= 1)

    kill_thread( node_execution_thread )

    return final_pos_reached
  end # insertion_compliant_move_urcap

  def insert_spiral_find_hole(axis = "Z", direction_sign = 1,
                              stop_force_threshold = 3,
                              max_radius = 0.005,
                              radius_incr_per_turn = 0.0003,
                              peck_mode = False,
                              tangential_speed = 0.005):

    if (stop_force_threshold < 0) or (stop_force_threshold > 40):
      popup("stop_force_threshold parameter in Newton must be between 0 and 40 Newtons","ERROR rq_insert_spiral_urcap")
      halt
    end
    if (max_radius < 0) or (max_radius > 0.05):
      popup("max_radius parameter must be between 0 mm and 50 mm","ERROR rq_insert_spiral_urcap")
      halt
    end
    if (radius_incr_per_turn < 0.00001) or (radius_incr_per_turn > 0.005):
      popup("radius_incr_per_turn parameter in mm must be between 0.01 mm and 5 mm","ERROR rq_insert_spiral_urcap")
      halt
    end

    rq_spiral_not_completed = False

    ins_x = 0
    ins_y = 0
    ins_z = 0
    ins_pose = p[0, 0, 0, 0, 0, 0]
    ins_current_pos = p[0, 0, 0, 0, 0, 0]
    ins_actual_angle = 0
    ins_search_result = False
    ins_radius_offset = 0
    ins_PI = 3.14159
    radius_inc_per_rad = radius_incr_per_turn / (2*ins_PI)
    ins_actual_radius = 0.0001  #Start radius
    ins_desired_arc_length = tangential_speed * rq_controller_time_step

    sleep(rq_controller_time_step)
    #Find the bore of the part
    ins_current_pos = get_actual_tcp_pose()
    sleep(rq_controller_time_step)

    # if axis == "Z"
    search_axis = 2
    other_axis_A = 0
    other_axis_B = 1
    if (axis == "X"):
      search_axis = 0
      other_axis_A = 1
      other_axis_B = 2
    elif (axis == "Y"):
      search_axis = 1
      other_axis_A = 2
      other_axis_B = 0
    end

    #********************************************************************************************************************
    #Spiral Search using any Axis
    #********************************************************************************************************************
    while ((ins_actual_radius <= max_radius) and (ins_actual_force_urcap(axis) >= stop_force_threshold)):
      if peck_mode:
        #Fragile mode, the robot rises between each new point
        #Retreat from position
        ins_pose[search_axis] = -0.002 * direction_sign
        next_tcp_pose = pose_trans(ins_current_pos,ins_pose)
        movej(next_tcp_pose)
        sleep(0.1)
        #Rotate
        ins_desired_arc_length = 0.0005
        delta_angle = ins_desired_arc_length / ins_actual_radius #small angle approximation
        ins_actual_angle = ins_actual_angle + delta_angle

        ins_pose[other_axis_A] = cos( ins_actual_angle ) * ins_actual_radius
        ins_pose[other_axis_B] = sin( ins_actual_angle ) * ins_actual_radius

        ins_actual_radius = ins_actual_angle * radius_inc_per_rad + ins_radius_offset
        next_tcp_pose = pose_trans(ins_current_pos, ins_pose)
        movej(next_tcp_pose)
        sleep(0.1)
        #Re-establish contact with the part
        ins_pose[search_axis] = 0.0005 * direction_sign
        next_tcp_pose = pose_trans(ins_current_pos, ins_pose)
        movel(next_tcp_pose, a=0.6, v=rq_ins_speed_setting)
        sleep(0.2)
      else:
        #standard mode: the Spiral_Search function will maintain contact between both mating parts at all times
        ins_pose[other_axis_A] = cos( ins_actual_angle ) * ins_actual_radius
        ins_pose[other_axis_B] = sin( ins_actual_angle ) * ins_actual_radius

        delta_angle = ins_desired_arc_length / ins_actual_radius
        ins_actual_angle = ins_actual_angle + delta_angle
        ins_actual_radius = ins_actual_angle * radius_inc_per_rad + ins_radius_offset
        next_tcp_pose = pose_trans(ins_current_pos,ins_pose)
        next_joint_pos = get_inverse_kin(next_tcp_pose)
        servoj(next_joint_pos, 0.1, 0.1, rq_controller_time_step, 0.05, 500)
      end
    end # while loop
    if (ins_actual_radius <= max_radius ):
      ins_search_result = True
    else:
      ins_search_result = False
      rq_spiral_not_completed = True
    end
    stopj(2)
    return ins_search_result

  end # insert_spiral_find_hole

  ####################  SPIRAL #############################
  def rq_insert_spiral_urcap(direction = "Z",
                             stop_force_threshold = 3,
                             max_radius = 0.005,
                             radius_incr = 0.0003,
                             peck_mode = False,
                             tangential_speed = 0.005,
                             compliant_insert_force_threshold = 10,
                             spiral_initial_pose_offset_name = "defaultname",
                             intelligent_approach_enabled = False):

    max_radius = max_radius / 1000 #TODO: change unit to meters and remove this line
    radius_incr = radius_incr / 1000 #TODO: change unit to meters and remove this line

    if (rq_insertion_force_node_id == -1):
      create_all_insertion_nodes()
    end

    hole_found = False
    spiral_bottom_target_reached = False
    number_of_failed_spiral_tries = 0
    number_of_spiral_tries_max = 5
    max_position_deviation = max_radius

    # define the direction sign from rq_ins_destination
    current_pose = get_actual_tcp_pose()
    rq_actual_to_destination = pose_trans(pose_inv(current_pose), rq_ins_destination)
    axis = str_at(direction, 0)
    direction_sign = 1
    direction = str_cat(axis,"+")
    if axis == "X":
      axis_index = 0
    elif axis == "Y":
      axis_index = 1
    elif axis == "Z":
      axis_index = 2
    else:
      textmsg("spiral insert, invalid direction ", direction)
    end
    if (rq_actual_to_destination[axis_index] < 0):
      direction_sign = -1
      direction = str_cat(axis,"-")
    end

    # linearsearch param
    lin_search_stop_force_threshold = compliant_insert_force_threshold
    spiral_initial_pose = get_actual_tcp_pose()
    if intelligent_approach_enabled:
      #adjust position using previous succesfull insertion final position
      spiral_initial_pose_offset = storevar.getvariablepose(spiral_initial_pose_offset_name, p[0,0,0,0,0,0])
      spiral_initial_pose_refined = pose_trans(spiral_initial_pose, spiral_initial_pose_offset)
      movel(spiral_initial_pose_refined, a = 0.1, v = 0.01)
      sleep(0.01)
    end
    while ( (spiral_bottom_target_reached == False) and (number_of_failed_spiral_tries < number_of_spiral_tries_max) ):
      rq_actual_to_destination = pose_trans(pose_inv(get_actual_tcp_pose()), rq_ins_destination)
      max_distance = norm( rq_actual_to_destination[axis_index] )
      contact_initiated = rq_linear_search_urcap(direction, lin_search_stop_force_threshold, tangential_speed, max_distance, 1)
      if contact_initiated:
        new_max_radius = determine_max_spiral_radius_from_actual_position(direction, spiral_initial_pose, max_radius)
        hole_found = insert_spiral_find_hole(axis, direction_sign, stop_force_threshold, new_max_radius, radius_incr, peck_mode, tangential_speed)
        if (hole_found == True): # if hole is found, try to insert
          max_force_control_position_deviation = determine_max_spiral_radius_from_actual_position(direction, spiral_initial_pose, max_radius)
          spiral_bottom_target_reached = insertion_compliant_move_urcap(axis, direction_sign, compliant_insert_force_threshold, tangential_speed, 1, max_force_control_position_deviation)
          if spiral_bottom_target_reached:
            if intelligent_approach_enabled:
              update_spiral_offset(direction, spiral_initial_pose, spiral_initial_pose_offset, spiral_initial_pose_offset_name) # update actual hole position.
            end
          else:
            textmsg("Insertion spiral: could not reach hole bottom")
          end
        else:
          textmsg("Insertion error: hole was not found after contact")
          break
        end
      else: # linear_search reached the teach position without contact
          spiral_bottom_target_reached = True
      end # if contact_initiated
      number_of_failed_spiral_tries = number_of_failed_spiral_tries + 1
    end # while
    return (not spiral_bottom_target_reached)
  end # rq_insert_spiral_urcap

  def insertion_finish_move_urcap(direction = "Z+"):
    insertion_offset = p[0,0,0,0,0,0]
    current_pose = get_actual_tcp_pose()
    rq_actual_to_destination = pose_trans(pose_inv(current_pose), rq_ins_destination)
    axis = str_at(direction, 0)
    if axis == "X":
      insertion_offset = p[rq_actual_to_destination[0],0,0,0,0,0]
    elif axis == "Y":
      insertion_offset = p[0,rq_actual_to_destination[1],0,0,0,0]
    elif axis == "Z":
      insertion_offset = p[0,0,rq_actual_to_destination[2],0,0,0]
    else:
      textmsg("insertion_finish_move_urcap, invalid direction ", direction)
    end
    insertion_pose = pose_trans(current_pose, insertion_offset)
    movel(insertion_pose, a=0.05, v=rq_ins_speed_setting)
  end

  def rq_xor(a, b):
    return (a and not(b)) or (not(a) and b)
  end

  def rq_adapt_force_control_to_direction(position_controlled_direction = 2, feature = 1, max_position_deviation = 0.1):
    force_control_enabled_vector = [True, True, True, False, False, False]
    force_control_enabled_vector[position_controlled_direction] = False
    targetForce = [0, 0, 0, 0, 0, 0]
    max_negative_deviation_vector = [-max_position_deviation, -max_position_deviation, -max_position_deviation, 0, 0, 0]
    max_positive_deviation_vector = [max_position_deviation, max_position_deviation, max_position_deviation, 0, 0, 0]
    max_negative_deviation_vector[position_controlled_direction] = 0
    max_positive_deviation_vector[position_controlled_direction] = 0
    adaptiveStiffness = True
    setup_force_node_on_server(rq_insertion_force_node_id,
                               feature, targetForce,
                               force_control_enabled_vector,
                               max_negative_deviation_vector,
                               max_positive_deviation_vector,
                               adaptiveStiffness)
  end

  def initialise_force_node(position_controlled_direction = 2, feature = 1, max_position_deviation = 0.1):
    movej(get_actual_joint_positions()) # This moveJ is used to prevent "another thread is already controlling the robot error".
    rq_adapt_force_control_to_direction(position_controlled_direction = position_controlled_direction,
                                        feature = 1,
                                        max_position_deviation = max_position_deviation)
    set_servoj_node_cmd(get_actual_joint_positions())
    reset_node_executor()
    active_and_reset_node(rq_insertion_force_node_id)
    active_and_reset_node(rq_insertion_servoj_node_id)
    node_execution_thread = run execute_node_thread()
    return node_execution_thread
  end

  ####################  ROTATIONAL #############################
  def rq_insert_rotation_urcap(positive_rotation_desired = True,
                               direction="Z",
                               speed = 0.004,
                               force_threshold = 10,
                               rotation_speed = 5,
                               max_angle_deg = 360,
                               peck_mode = False,
                               max_rotation_torque=1):

    speed = speed / 1000 # TODO: change speed input units to meters instead of mm and remove this line
    max_force_control_position_deviation = 0.002 # TODO: add a parameter for this in the interface
    max_torque_reached_counter_fail_threshold = 1/rq_controller_time_step # try for about one second

    if (rq_insertion_force_node_id == -1):
        create_all_insertion_nodes()
    end

    # define the direction sign
    rq_actual_to_destination = pose_trans(pose_inv(get_actual_tcp_pose()), rq_ins_destination)
    axis = str_at(direction, 0)
    direction_sign = 1
    direction = str_cat(axis,"+")
    if axis == "X":
      rq_ins_offset = p[rq_actual_to_destination[0], 0, 0, 0, 0, 0]
      rot_axe = 3
      axis_index = 0
    elif axis == "Y":
      rq_ins_offset = p[0, rq_actual_to_destination[1], 0, 0, 0, 0]
      rot_axe = 4
      axis_index = 1
    elif axis == "Z":
      rq_ins_offset = p[0, 0, rq_actual_to_destination[2], 0, 0, 0]
      rot_axe = 5
      axis_index = 2
    else:
      textmsg("insertion: invalid direction ", direction)
    end
    if (rq_actual_to_destination[axis_index] < 0):
      direction_sign = -1
      direction = str_cat(axis,"-")
      positive_rotation_desired = not positive_rotation_desired
    end

    distance_to_destination = norm( rq_actual_to_destination[axis_index] )

    contact_with_piece_initiated = rq_linear_search_urcap(direction, force_threshold, speed, distance_to_destination, feature = 1)

    if( contact_with_piece_initiated ):

      # verify validity of user inputs
      if ((rotation_speed <= 0) or (rotation_speed > 60)):
        popup("rotation speed parameter in degrees / second must be between 0.01 and 60","ERROR rq_insert_rotation_urcap")
        halt
      elif ((max_rotation_torque < 0.01) or (max_rotation_torque > 15)):
        popup("max_rotation_torque parameter in Newton-meter must be between 0.01 and 15","ERROR rq_insert_rotation_urcap")
        halt
      elif ((max_angle_deg <= 1) or (max_angle_deg > 360)):
        popup("max angle parameter in degree must be between 1 and 360","ERROR rq_insert_rotation_urcap")
        halt
      end

      # initialize forcenode: adapt to direction
      node_execution_thread = initialise_force_node(position_controlled_direction = axis_index,
                                                    feature = 1,
                                                    max_position_deviation = max_force_control_position_deviation)

      if positive_rotation_desired:
        rot_direction_sign = 1
      else:
        rot_direction_sign = -1
      end
      rq_ins_speed_setting = speed
      posrot = p[0,0,0,0,0,0]
      max_rot_angle = d2r(max_angle_deg)
      time_step_signed = rq_controller_time_step * rot_direction_sign * direction_sign
      rot_step = d2r(rotation_speed) * time_step_signed
      rot_step_5deg_per_second = d2r(5) * time_step_signed

      line_step = rq_ins_speed_setting * rq_controller_time_step * direction_sign
      rot_actual_angle = 0
      rot_actual_mode = 1 #1= linear, 2 = rotation
      rot_actual_distance = 0
      ins_rotation_initial_pose = get_actual_tcp_pose()
      rq_actual_to_destination = pose_trans( pose_inv(ins_rotation_initial_pose), rq_ins_destination )
      distance_to_destination = norm( rq_actual_to_destination[axis_index] )
      global rq_insertion_max_torque_reached_counter = 0

      if peck_mode:
        #peck mode
        positive_rotation_computed = positive_rotation_desired
        while ( (norm(rot_actual_distance) < distance_to_destination) and
                (norm(rot_actual_angle) <= max_rot_angle) and
                (rq_insertion_max_torque_reached_counter < max_torque_reached_counter_fail_threshold) ):
          is_max_torque_reached = norm(get_applied_tcp_force(rot_axe)) > max_rotation_torque
          if (ins_actual_force_urcap(direction) >= force_threshold):
            #goes up
            posrot[axis_index] = rot_actual_distance - 0.002 * direction_sign
            next_tcp_pose = pose_trans(ins_rotation_initial_pose, posrot)
            next_joint_pos = get_inverse_kin(next_tcp_pose)
            node_rpc_server.movejdefinewaypoint(rq_insertion_movej_node_id, next_joint_pos, 0.4, 0.4)
            execute_node(rq_insertion_movej_node_id, False )
            #rotate
            rot_actual_angle = compute_rotation_next_angle(rot_actual_angle, 285 * rot_step, is_max_torque_reached) # value of 285 define the peck mode "step size". determined ad oc
            posrot[rot_axe] = rot_actual_angle
            next_tcp_pose = pose_trans(ins_rotation_initial_pose, posrot)
            next_joint_pos = get_inverse_kin(next_tcp_pose)
            node_rpc_server.movejdefinewaypoint(rq_insertion_movej_node_id, next_joint_pos, 1, 1)
            execute_node(rq_insertion_movej_node_id, False )
            #go back in touch with the part
            posrot[axis_index] = rot_actual_distance
            next_tcp_pose = pose_trans(ins_rotation_initial_pose, posrot)
            next_joint_pos = get_inverse_kin(next_tcp_pose)
            node_rpc_server.movejdefinewaypoint(rq_insertion_movej_node_id, next_joint_pos, 0.4, 0.3)
            execute_node(rq_insertion_movej_node_id, False )
            sleep(0.1)
          else:
            rq_insertion_max_torque_reached_counter = 0
            rot_actual_distance = rot_actual_distance + line_step
            posrot[axis_index] = rot_actual_distance
            next_tcp_pose = pose_trans(ins_rotation_initial_pose, posrot)
            next_joint_pos = get_inverse_kin(next_tcp_pose)
            update_servoj_node_target(next_joint_pos)
            if (rq_active_node != rq_insertion_servoj_node_id):
              active_and_reset_node(rq_insertion_servoj_node_id)
            end
          end # if
        end # while
      else:
        #normal mode
        while ( (norm(rot_actual_distance) <= distance_to_destination) and
                (norm(rot_actual_angle) <= max_rot_angle) and
                (rq_insertion_max_torque_reached_counter < max_torque_reached_counter_fail_threshold) ):
          is_max_torque_reached = norm(get_applied_tcp_force(rot_axe)) > max_rotation_torque
          if ( norm(get_applied_tcp_force(axis_index)) >= force_threshold ):
            if (rot_actual_mode == 1):
              rot_actual_distance = rot_actual_distance - line_step
              posrot[axis_index] = rot_actual_distance
            end
            limited_rotation_step = limit_rotation_step_when_close_to_max_angle(rot_step, rot_step_5deg_per_second, max_rot_angle, rot_actual_angle)
            rot_actual_angle = compute_rotation_next_angle(rot_actual_angle, limited_rotation_step, is_max_torque_reached)
            posrot[rot_axe] = rot_actual_angle
            rot_actual_mode = 2
          else:
            rq_insertion_max_torque_reached_counter = 0
            rot_actual_distance = rot_actual_distance + line_step
            posrot[axis_index] = rot_actual_distance
            rot_actual_mode = 1
          end # if
          next_tcp_pose = pose_trans(ins_rotation_initial_pose, posrot)
          next_joint_pos = get_inverse_kin(next_tcp_pose)
          update_servoj_node_target(next_joint_pos)
        end # while
      end # if peck_mode

      kill_thread( node_execution_thread )
      stopj(2)
      rq_rotation_not_completed = ( (norm(rot_actual_angle) > max_rot_angle) or
                                    (rq_insertion_max_torque_reached_counter >= max_torque_reached_counter_fail_threshold) )
    else: # initial find_surface was unsuccessfull, assume a direct hit to target, which is a success
      rq_rotation_not_completed = False
    end # if contact_with_piece_initiated

    return rq_rotation_not_completed
  end # insert rotation 2

  def limit_rotation_step_when_close_to_max_angle(rot_step, minimal_rot_step, max_rot_angle, rot_actual_angle):
    rot_deceleration_angle_distance = d2r(3)
    rot_direction = 1
    if( rot_step < 0 ):
      rot_direction = -1
      rot_step = -1 * rot_step # get positive rot_step for calculation. Direction sign is re-introduced at the end.
    end
    angle_distance_to_max_rot_angle = max_rot_angle - norm(rot_actual_angle)
    if( (angle_distance_to_max_rot_angle < rot_deceleration_angle_distance) and (rot_step > minimal_rot_step) ):
      decelaration_slope = (rot_step - minimal_rot_step) / rot_deceleration_angle_distance
      rot_step_limited = decelaration_slope * angle_distance_to_max_rot_angle + minimal_rot_step
    else:
      rot_step_limited = rot_step
    end
    return ( rot_direction * rot_step_limited )
  end

  def compute_rotation_next_angle(current_angle, step, is_max_torque_reached):
  #This function compute the rotation angle for rotational insertion by
  # incrementing the current angle by the desired step size.
  # If the maximal torque is reached, the rotation goes backward to
  # return to a admissible torque. In the backward direction,
  # a smaller step size is used to prevent constant oscillation between to steps
    if (is_max_torque_reached):
        rq_insertion_max_torque_reached_counter = rq_insertion_max_torque_reached_counter + 1
        new_angle = current_angle - 0.8 * step
    else:
        new_angle = current_angle + step
    end
    return new_angle
  end

  def center_one_axis(axis, lin_search_stop_force_threshold, speed, max_distance, feature):
    # Initiate contact in forward direction
    contact_initiated = rq_linear_search_urcap( str_cat(axis, "+"), lin_search_stop_force_threshold, speed, max_distance, feature)
    if contact_initiated:
      forward_contact_pose = get_actual_tcp_pose()
      # Initiate contact in reverse direction
      contact_initiated = rq_linear_search_urcap(str_cat(axis, "-"), lin_search_stop_force_threshold, speed, max_distance, feature)
      if contact_initiated:
        reverse_contact_pose = get_actual_tcp_pose()
        # Go to average of contact points
        pose_center_1 = interpolate_pose(forward_contact_pose, reverse_contact_pose, 0.5)
        movel(pose_center_1, a=0.6, v=speed)
      end
    end
    return contact_initiated
  end

  def rq_insert_recenter_urcap(axis = "Z", max_distance = 0.1, speed = 0.005, feature = 1, lin_search_stop_force_threshold = 5):

    if (max_distance < 0) or (max_distance > 1):
      popup("max_distance parameter in m must be between 0 and 1","ERROR rq_insert_recenter_urcap")
      halt
    elif (speed < 0.0001) or (speed > 0.5):
      popup("max_radius parameter in mm must be between 0.0001m/s and 0.5m/s","ERROR rq_insert_recenter_urcap")
      halt
    end

    #--------------------------------------------------------------------------------------------------------------------
    #For insertion in the X axis
    #--------------------------------------------------------------------------------------------------------------------
    if (axis == "X"):
      recenter_axis_1 = "Y"
      recenter_axis_2 = "Z"
    #--------------------------------------------------------------------------------------------------------------------
    #For insertion in the Y axis
    #--------------------------------------------------------------------------------------------------------------------
    elif (axis == "Y"):
      recenter_axis_1 = "X"
      recenter_axis_2 = "Z"
    #--------------------------------------------------------------------------------------------------------------------
    #For insertion in the Z axis
    #--------------------------------------------------------------------------------------------------------------------
    elif (axis == "Z"):
      recenter_axis_1 = "X"
      recenter_axis_2 = "Y"
    end

    recenter_successfull = center_one_axis(recenter_axis_1, lin_search_stop_force_threshold, speed, max_distance, feature)
    if recenter_successfull:
      recenter_successfull = center_one_axis(recenter_axis_2, lin_search_stop_force_threshold, speed, max_distance, feature)
    end

    if (recenter_successfull == False):
      textmsg("rq_insert_recenter_urcap failed, could not initiate contact with piece")
    end

    return recenter_successfull
  end # rq_insert_recenter_urcap

  # ******************* MAIN of Insertion Preamble *******************
  storevar.clearall()
  global rq_insertion_force_node_id = -1
  def rq_linear_search_common_validation(abs_max_distance, speed, force_threshold):
    if (abs_max_distance > 2.0):
      popup("maximum distance parameter in meters must be between 0 and 2.0","ERROR rq_linear_search_urcap")
      halt
    elif (speed < 0.0001) or (speed > 0.15):
      popup("speed parameter in mm/s must be between 0.1 and 150","ERROR rq_linear_search_urcap")
      halt
    elif (force_threshold < 0.0) or (force_threshold > 200):
      popup("Force parameter in Newtons must be between 0 and 200","ERROR rq_linear_search_urcap")
      halt
    end
  end

  def rq_linear_search_get_direction_sign(direction):
    sign = str_at(direction, 1)
    direction_sign = 1
    if sign == "-":
      direction_sign = -1
    end
    return direction_sign
  end

  def rq_linear_search_get_force_index(direction):
    axis = str_at(direction, 0)
    force_index = 0
    if (axis == "X") or (axis == "x"):
      force_index = 0
    elif (axis == "Y") or (axis == "y"):
      force_index = 1
    elif (axis == "Z") or (axis == "z"):
      force_index = 2
    else:
      popup("direction parameter must be X+, X-, Y+, Y-, Z+ or Z-","ERROR rq_linear_search_urcap")
      halt
    end
    return force_index
  end

  def rq_linear_search_get_pose_offset(force_index, max_distance):
    pose_offset = p[0,0,0,0,0,0]
    pose_offset[force_index] = max_distance
    return pose_offset
  end

  def rq_linear_search_execution(pose_from, pose_to, force_threshold, speed, T_tcp_to_force_frame, force_index, direction_sign):
    steptime = rq_controller_time_step
    distance = point_dist(pose_from, pose_to)
    number_pose_interpolate = floor(distance / (speed * steptime)) + 1
    delta_alpha = 1.0 / number_pose_interpolate

    alpha = 0.0
    local surface_found = False

    pose_step = 0
    end_pose_pause_time = 0.2 # to refine
    max_pose_steps = number_pose_interpolate + end_pose_pause_time/steptime
    while (pose_step < max_pose_steps) and (not surface_found):
      pose_step = pose_step + 1
      alpha = pose_step * delta_alpha
      if (alpha < 1.0):
        pose_interpolate = interpolate_pose(pose_from, pose_to, alpha)
      else:
        pose_interpolate = pose_to
      end

      servoj(get_inverse_kin(pose_interpolate), 0.1, 0.1, steptime, 0.05, 500)

      wrench = express_force_in_frame(T_tcp_to_force_frame, tcp_wrench)
      applied_force = -1 * wrench[force_index]

      if (direction_sign * applied_force) >= force_threshold:
        surface_found = True
      end
    end

    return surface_found
  end

  #************************************************
  #Function:  rq_linear_search_urcap(direction="Z+", force[N] = 10, speed[m/s] = 0.004, max_distance[m] = 0.02)
  #   Find a specific force in the direction of "direction".
  #   Robot will move towards a max_distance from the current position in the tool frame
  #   Return True if the force is detected during the robot motion
  #
  #************************************************
  def rq_linear_search_urcap(direction="Z+", force_threshold = 10, speed = 0.004, max_distance = 0.02, feature = 0 ):

    rq_linear_search_common_validation(max_distance, speed, force_threshold)
    if (feature != 0) and (feature != 1):
      popup("feature value should be 0 for base or 1 for tool","ERROR rq_linear_search_urcap")
      halt
    end

    feature_base = 0
    feature_tool = 1

    force_index = rq_linear_search_get_force_index(direction)
    direction_sign = rq_linear_search_get_direction_sign(direction)
    max_distance = direction_sign * max_distance
    pose_offset = rq_linear_search_get_pose_offset(force_index, max_distance)

    tcp_pose = get_actual_tcp_pose()
    pose_from = tcp_pose
    pose_to = pose_from
    if feature == feature_base:
      pose_to = pose_add(pose_from, pose_offset)
    elif feature == feature_tool:
      pose_to = pose_trans(pose_from, pose_offset)
    end

    T_tcp_to_force_frame = p[0, 0, 0, 0, 0, 0] # default for feature_tool
    if (feature == feature_base):
      T_tcp_to_force_frame = pose_inv(tcp_pose)
    end

    surface_found = rq_linear_search_execution(pose_from, pose_to, force_threshold, speed, T_tcp_to_force_frame, force_index, direction_sign)

    return surface_found
  end

  def rq_linear_search_custom_frame(direction="Z+", force_threshold = 10, speed = 0.004, abs_max_distance = 0.02, feature_frame = p[0, 0, 0, 0, 0, 0]):

    rq_linear_search_common_validation(abs_max_distance, speed, force_threshold)

    force_index = rq_linear_search_get_force_index(direction)
    direction_sign = rq_linear_search_get_direction_sign(direction)
    max_distance = direction_sign * abs_max_distance
    pose_offset = rq_linear_search_get_pose_offset(force_index, max_distance)

    tcp_pose = get_actual_tcp_pose()
    offset_frame = p[tcp_pose[0], tcp_pose[1], tcp_pose[2], feature_frame[3], feature_frame[4], feature_frame[5]]
    tcp_position_with_offset = pose_trans(offset_frame, pose_offset)
    pose_from = tcp_pose
    pose_to = p[tcp_position_with_offset[0], tcp_position_with_offset[1], tcp_position_with_offset[2], tcp_pose[3], tcp_pose[4], tcp_pose[5]]

    T_tcp_to_force_frame = pose_trans(pose_inv(tcp_pose), feature_frame)

    surface_found = rq_linear_search_execution(pose_from, pose_to, force_threshold, speed, T_tcp_to_force_frame, force_index, direction_sign)

    return surface_found
  end

  def validate_wait_for_force_drop_common_parameters(force_threshold, timeout_seconds):
    if (timeout_seconds < 0.0) or (timeout_seconds > 3600):
      popup("timeout parameter in s must be between 0 and 3600","ERROR rq_wait_for_force_drop")
      halt
    elif (force_threshold < 0.0) or (force_threshold > 200):
      popup("Force parameter in Newtons must be between 0 and 200","ERROR rq_wait_for_force_drop")
      halt
    end
  end

  def rq_wait_for_force_drop_execution(force_threshold, T_tcp_to_force_frame, force_index, direction_sign, timeout_seconds):
    local steptime = get_steptime()
    local release_detected = False
    local time = 0

    while (time < timeout_seconds) and (not release_detected):
      time = time + steptime

      local wrench = express_force_in_frame(T_tcp_to_force_frame, tcp_wrench)
      local force = -1 * wrench[force_index]

      if (direction_sign * force) < force_threshold:
        release_detected = True
      end
      sync()
    end

    return release_detected
  end

  def rq_wait_for_force_drop_custom_frame(direction="Z+", force_threshold = 10, timeout_seconds = 60, feature_frame = p[0, 0, 0, 0, 0, 0] ):
    validate_wait_for_force_drop_common_parameters(force_threshold, timeout_seconds)

    local force_index = rq_linear_search_get_force_index(direction)
    local direction_sign = rq_linear_search_get_direction_sign(direction)

    local tcp_pose = get_actual_tcp_pose()
    local T_tcp_to_force_frame = pose_trans(pose_inv(tcp_pose), feature_frame)

    local release_detected = rq_wait_for_force_drop_execution(force_threshold, T_tcp_to_force_frame, force_index, direction_sign, timeout_seconds)

    return release_detected
  end

  def rq_wait_for_force_drop(direction="Z+", force_threshold = 10, timeout_seconds = 60, feature = 0 ):
    validate_wait_for_force_drop_common_parameters(force_threshold, timeout_seconds)
    if (feature != 0) and (feature != 1):
      popup("feature value should be 0 for base or 1 for tool","ERROR rq_wait_for_force_drop")
      halt
    end

    local force_index = rq_linear_search_get_force_index(direction)
    local direction_sign = rq_linear_search_get_direction_sign(direction)

    local feature_base = 0
    local feature_tool = 1
    local tcp_pose = get_actual_tcp_pose()
    local T_tcp_to_force_frame = p[0, 0, 0, 0, 0, 0] # default for feature_tool
    if (feature == feature_base):
      T_tcp_to_force_frame = pose_inv(tcp_pose)
    end

    local release_detected = rq_wait_for_force_drop_execution(force_threshold, T_tcp_to_force_frame, force_index, direction_sign, timeout_seconds)

    return release_detected
  end



    ##############################################
    # OFFSET FEATURE-RELATED VARIABLES AND METHODS
    ##############################################
    def cross_product(vector1,vector2):
      v_temp=[0,0,0]
      v_temp[0]=vector1[1]*vector2[2]-vector1[2]*vector2[1]
      v_temp[1]=vector1[2]*vector2[0]-vector1[0]*vector2[2]
      v_temp[2]=vector1[0]*vector2[1]-vector1[1]*vector2[0]
      return v_temp
    end

    def relocate_xyzr(init_feature, init_touch_pose, touch_pose):
      init_touch_pose_2_init_feature = pose_trans( pose_inv(init_touch_pose), init_feature)
      new_feature = pose_trans( touch_pose, init_touch_pose_2_init_feature )

      return new_feature
    end

    def relocate_orientation(touch1_init_pose, touch2_init_pose, feature_init_pose, touch1_pose, touch2_pose):
      #when relocating using 2 touch, the center of rotation is around touch point 1 (this could be changed)

      # initial touch2 pose in initial touch 1 pose frame:
      touch2_initial_pose_in_touch1_initial_pose_frame = pose_trans(pose_inv(touch1_init_pose), touch2_init_pose)

      # find theoric touch2_pose if no rotation
      touch2_pose_if_no_rotation = pose_trans(touch1_pose, touch2_initial_pose_in_touch1_initial_pose_frame)

      # vectors touch1 to touch2
      touch1_pose_to_touch2_pose = pose_trans(pose_inv(touch1_pose), touch2_pose)
      touch1_pose_to_touch2_pose_if_no_rotation = pose_trans(pose_inv(touch1_pose), touch2_pose_if_no_rotation)

      #angle axis calculation
      normal_vector = cross_product(touch1_pose_to_touch2_pose_if_no_rotation, touch1_pose_to_touch2_pose)
      normal_vector_norm = norm(normal_vector)
      if (normal_vector_norm > 10e-6):
        rotation_angle_rad = asin( normal_vector_norm / (norm(touch1_pose_to_touch2_pose_if_no_rotation) * norm(touch1_pose_to_touch2_pose) ) )
        normal_vector_to_angle_axis_multiply_norm_factor = rotation_angle_rad / normal_vector_norm
        angle_axis = [normal_vector[0] * normal_vector_to_angle_axis_multiply_norm_factor, normal_vector[1] * normal_vector_to_angle_axis_multiply_norm_factor, normal_vector[2] * normal_vector_to_angle_axis_multiply_norm_factor]
        rotation_offset_pose = p[0, 0, 0, angle_axis[0], angle_axis[1], angle_axis[2]]

        #rotate touch1 pose using touch2 information
        touch1_pose_rotated = pose_trans(touch1_pose, rotation_offset_pose)
      else:
        touch1_pose_rotated = touch1_pose
      end

      # relocate the feature using touch1_rotated_pose
      return relocate_xyzr(feature_init_pose, touch1_init_pose, touch1_pose_rotated)
    end

    def relocate_1_touch(touch_init_pose, touch_pose, feature_init_pose, feature_actual_pose):
      touch_initial_pose_in_initial_feature_frame = pose_trans(pose_inv(feature_init_pose), touch_init_pose)
      touch_actual_pose_in_actual_feature_frame = pose_trans(pose_inv(feature_actual_pose), touch_pose)

      # difference between touch poses in their respective feature frame
      touch_pose_offset = pose_sub(touch_actual_pose_in_actual_feature_frame, touch_initial_pose_in_initial_feature_frame)

      # remove all rotation from offset
      touch_pose_offset[3] = 0
      touch_pose_offset[4] = 0
      touch_pose_offset[5] = 0

      # apply pose offset to actual feature
      return pose_trans(feature_actual_pose, touch_pose_offset)
    end
    ##############################################
    # PALLETIZER INITIALIZATION
    ##############################################
    global rq_palletizer_state_changed = False

    def assert_not_in_palletizer_node(function_name):
      rq_palletizer_uuid = palletizerXmlRpcClient.getCurrentPalletizerNode()
      if (rq_palletizer_uuid != ""):
        popup(str_cat(function_name," should never be called from within a Palletizer node."), title="Palletizer", error=True, blocking=True)
        halt
      end
    end

    # Documented in monorepo/doc/pal/PalAdvancedProgrammingFunctions.md
    def rq_pallet_viewer(runtime=True):

      assert_not_in_palletizer_node("rq_pallet_viewer")

      if(not palletizerXmlRpcClient.acknowledgePalletStates(runtime)):
        checkForScriptPreparationException()
        halt
      end

      if (runtime):
        rq_palletizer_state_changed = True
      end
    end

    palletizerXmlRpcClient.setCurrentPalletizerNode("")

    rq_pallet_viewer(runtime=False)


    ##############################################
    # PALLETIZER-RELATED VARIABLES AND METHODS
    ##############################################

    # Documented in monorepo/doc/pal/PalAdvancedProgrammingFunctions.md
    def rq_get_nb_processed_boxes():
      rq_palletizer_uuid = palletizerXmlRpcClient.getCurrentPalletizerNode()
      if rq_palletizer_uuid == "":
        popup("rq_get_nb_processed_boxes() should only be called from within a Palletizer node.", title="Palletizer", error=True, blocking=True)
        halt
      end

      rq_box_count = palletizerXmlRpcClient.getCurrentBoxCount(rq_palletizer_uuid)
      if rq_box_count == -1:
        popup("Invalid Palletizer node id used for rq_get_nb_processed_boxes()", title="Palletizer", error=True, blocking=True)
        halt
      end
      return rq_box_count
    end

    # Documented in monorepo/doc/pal/PalAdvancedProgrammingFunctions.md
    def rq_get_current_box_type():
         rq_palletizer_uuid = palletizerXmlRpcClient.getCurrentPalletizerNode()
         if rq_palletizer_uuid == "":
            popup("rq_get_current_box_type() should only be called from within a Palletizer node.", title="Palletizer", error=True, blocking=True)
            halt
         end

         rq_box_type_name = palletizerXmlRpcClient.getCurrentBoxTypeName(rq_palletizer_uuid)
         return rq_box_type_name
    end

    # Documented in monorepo/doc/pal/PalAdvancedProgrammingFunctions.md
    def rq_get_current_pal_recipe():
        rq_palletizer_uuid = palletizerXmlRpcClient.getCurrentPalletizerNode()
        if rq_palletizer_uuid == "":
           popup("rq_get_current_pal_recipe() should only be called from within a Palletizer node.", title="Palletizer", error=True, blocking=True)
           halt
        end

        rq_pal_unit_load_name = palletizerXmlRpcClient.getCurrentPalletUnitLoadName(rq_palletizer_uuid)
        return rq_pal_unit_load_name
    end

    # Documented in monorepo/doc/pal/PalAdvancedProgrammingFunctions.md
    def rq_set_pallet_completed():
      rq_palletizer_uuid = palletizerXmlRpcClient.getCurrentPalletizerNode()
      if rq_palletizer_uuid == "":
        popup("rq_set_pallet_completed() should only be called from within a Palletizer node.", title="Palletizer", error=True, blocking=True)
        halt
      end

      palletizerXmlRpcClient.skipToAfterPallet(rq_palletizer_uuid)
    end

    # Documented in monorepo/doc/pal/PalAdvancedProgrammingFunctions.md
    def rq_demo_mode_switch_palletizer_mode():
      palletizerXmlRpcClient.demoModeFakePalletSwapAndAndSwitchPalletizerMode()
    end

    def rq_linear_axis_scan(halt_on_error=True):
      local succeeded = False
      local error_message = ""

      if not node_rpc_server.linearaxisconnected():
        succeeded = node_rpc_server.linearaxisscan()
        if succeeded:
          textmsg("Linear axis scanned successfully")
        else:
          error_message = "rq_linear_axis_scan() was unable to find linear axis"
        end
      else:
        succeeded = True
        textmsg("Linear axis already connected")
      end

      if not succeeded:
        if halt_on_error:
          popup(error_message, title="Linear Axis", error=True, blocking=True)
          halt
        else:
          textmsg(error_message)
        end
      end

      return succeeded
    end

    # Documented in monorepo/doc/pal/PalAdvancedProgrammingFunctions.md
    def rq_linear_axis_start(halt_on_error=True):
      local succeeded = False
      local error_message = ""

      if not node_rpc_server.linearaxisconnected():
        error_message = "rq_linear_axis_start() was unable to start linear axis : linear axis not connected"
      else:
        succeeded = node_rpc_server.linearaxisstart()
        if succeeded:
          textmsg("Linear axis started successfully")
        else:
          error_message = "rq_linear_axis_start() was unable to start linear axis"
        end
      end

      if not succeeded:
        if halt_on_error:
          popup(error_message, title="Linear Axis", error=True, blocking=True)
          halt
        else:
          textmsg(error_message)
        end
      end

      return succeeded
    end

    # Documented in monorepo/doc/pal/PalAdvancedProgrammingFunctions.md
    def rq_linear_axis_disable(halt_on_error=True):
      local succeeded = False
      local error_message = ""

      if not node_rpc_server.linearaxisconnected():
        error_message = "rq_linear_axis_disable() was unable to disable linear axis : linear axis not connected"
      else:
        succeeded = node_rpc_server.linearaxisdisable()
        if succeeded:
          textmsg("Linear axis disabled successfully")
        else:
          error_message = "rq_linear_axis_disable() was unable to disable linear axis"
        end
      end

      if not succeeded:
        if halt_on_error:
          popup(error_message, title="Linear Axis", error=True, blocking=True)
          halt
        else:
          textmsg(error_message)
        end
      end

      return succeeded
    end

    # Documented in monorepo/doc/pal/PalAdvancedProgrammingFunctions.md
    def rq_set_palletizer_state(palletizer_index, processed_boxes, next_step, other_pallet_state="ABSENT", current_pallet="CURRENT", left_recipe="", right_recipe=""):
      assert_not_in_palletizer_node("rq_set_palletizer_state")

      palletizerXmlRpcClient.setPalletizerState(palletizer_index, processed_boxes, next_step, other_pallet_state, current_pallet, left_recipe, right_recipe)
      checkForScriptPreparationException()
      rq_palletizer_state_changed = True
    end

    # Documented in monorepo/doc/pal/PalAdvancedProgrammingFunctions.md
    def rq_get_pallet_state(is_pallet_left):
      return node_rpc_server.getPalletState(is_pallet_left)
    end

    # Documented in monorepo/doc/pal/PalAdvancedProgrammingFunctions.md
    def rq_use_payload_with_box(ratio=1):
      local rq_palletizer_uuid = palletizerXmlRpcClient.getCurrentPalletizerNode()
      if rq_palletizer_uuid == "":
        popup("rq_use_payload_with_box() should only be called from within a Palletizer node.", title="Palletizer", error=True, blocking=True)
        halt
      end

      if ratio < 0 or ratio > 1:
        popup("rq_use_payload_with_box: ratio should be in range [0, 1].", title="Palletizer", error=True, blocking=True)
        halt
      end

      local initial_payload = palletizerXmlRpcClient.getInitialPayload()
      local initial_center_of_gravity = palletizerXmlRpcClient.getInitialCenterOfGravity()
      local box_payload = palletizerXmlRpcClient.getCurrentBoxTypeWeight(rq_palletizer_uuid) * ratio
      local tcp_offset_from_flange = get_tcp_offset()
      local current_box_type_cog_offset = palletizerXmlRpcClient.getCurrentBoxTypeCenterOfGravityInTcpreferenceFrame(rq_palletizer_uuid)
      local current_box_type_cog_in_tcp_frame  = p[
        current_box_type_cog_offset[0],
        current_box_type_cog_offset[1],
        current_box_type_cog_offset[2],
        0, 0, 0
      ]
      local box_center_of_gravity_in_flange_reference_frame = pose_trans(tcp_offset_from_flange, current_box_type_cog_in_tcp_frame)
      local new_payload = initial_payload + box_payload
      if new_payload > 0:
         local new_center_of_gravity = [
            (initial_center_of_gravity[0]*initial_payload + box_center_of_gravity_in_flange_reference_frame[0]*box_payload) / new_payload,
            (initial_center_of_gravity[1]*initial_payload + box_center_of_gravity_in_flange_reference_frame[1]*box_payload) / new_payload,
            (initial_center_of_gravity[2]*initial_payload + box_center_of_gravity_in_flange_reference_frame[2]*box_payload) / new_payload
         ]
         set_target_payload(new_payload, new_center_of_gravity)
      end
      palletizerXmlRpcClient.setPayloadModifiedByScriptFunction()
    end

    def rq_use_payload_without_box():
      local rq_palletizer_uuid = palletizerXmlRpcClient.getCurrentPalletizerNode()
      if rq_palletizer_uuid == "":
        popup("rq_use_payload_without_box() should only be called from within a Palletizer node.", title="Palletizer", error=True, blocking=True)
        halt
      end

      local initial_payload = palletizerXmlRpcClient.getInitialPayload()
      local initial_center_of_gravity = palletizerXmlRpcClient.getInitialCenterOfGravity()
      set_target_payload(initial_payload, initial_center_of_gravity)
      palletizerXmlRpcClient.setPayloadModifiedByScriptFunction()
    end

    # Documented in monorepo/doc/pal/PalAdvancedProgrammingFunctions.md
    def rq_use_payload_no_box():
      rq_use_payload_without_box()
    end

    # Documented in monorepo/doc/pal/PalAdvancedProgrammingFunctions.md
    def rq_set_box_payload(box_payload):
      local rq_palletizer_uuid = palletizerXmlRpcClient.getCurrentPalletizerNode()
      if rq_palletizer_uuid == "":
        popup("rq_set_box_payload(box_payload) should only be called from within a Palletizer node.", title="Palletizer",
        error=True, blocking=True)
        halt
      end

      if box_payload < 0 or box_payload > 20:
        popup("rq_set_box_payload: box payload should be between 0 and 20 kg.", title="Palletizer", error=True, blocking=True)
        halt
      end

      palletizerXmlRpcClient.setCurrentBoxTypeWeight(rq_palletizer_uuid, box_payload)
    end

    # Documented in monorepo/doc/pal/PalAdvancedProgrammingFunctions.md
    def rq_register_bounding_box(referential, position, dimensions):
      local rq_pose_string = str_cat("", position)
      rq_pose_string = str_sub(rq_pose_string, 1, str_len(rq_pose_string))

      local rq_json_string = str_cat("{'boundingBoxes':[{'parentId':", referential)
      rq_json_string = str_cat(rq_json_string, ", 'pose':")
      rq_json_string = str_cat(rq_json_string, rq_pose_string)
      rq_json_string = str_cat(rq_json_string, ",'dimensions':")
      rq_json_string = str_cat(rq_json_string, dimensions)
      rq_json_string = str_cat(rq_json_string, "}]}")

      node_rpc_server.configurePalletizerInstallation(rq_json_string)
    end

    # Documented in monorepo/doc/pal/PalAdvancedProgrammingFunctions.md
    def rq_set_gripper_collision_model(fileName, referenceFrame, filePath="/programs/"):
        local rq_json_string = str_cat("{'gripperMesh':{'fileName':'", fileName)
        rq_json_string = str_cat(rq_json_string, "', 'filePath':'")
        rq_json_string = str_cat(rq_json_string, filePath)
        rq_json_string = str_cat(rq_json_string, "','referenceFrame':")
        rq_json_string = str_cat(rq_json_string, referenceFrame)
        rq_json_string = str_cat(rq_json_string, "}}")

        node_rpc_server.configurePalletizerInstallation(rq_json_string)
    end

